C09150=1155.130,217.101,-63.506,-177.845,7.375,148.764
C09151=1155.134,216.851,-63.482,-177.849,7.372,148.764
C09152=1155.139,216.603,-63.456,-177.851,7.369,148.764
C09153=1155.143,216.355,-63.430,-177.854,7.367,148.765
C09154=1155.148,216.106,-63.406,-177.857,7.365,148.765
C09155=1155.152,215.857,-63.380,-177.860,7.362,148.765
C09156=1155.157,215.609,-63.356,-177.862,7.360,148.765
C09157=1155.161,215.360,-63.330,-177.865,7.357,148.765
C09158=1155.166,215.111,-63.306,-177.867,7.355,148.766
C09159=1155.170,214.862,-63.280,-177.871,7.352,148.766
C09160=1155.175,214.614,-63.256,-177.873,7.349,148.766
C09161=1155.179,214.364,-63.231,-177.876,7.347,148.766
C09162=1155.184,214.116,-63.205,-177.879,7.345,148.766
C09163=1155.188,213.867,-63.181,-177.881,7.343,148.767
C09164=1155.193,213.619,-63.156,-177.884,7.340,148.767
C09165=1155.197,213.370,-63.130,-177.887,7.337,148.767
C09166=1155.202,213.121,-63.106,-177.889,7.335,148.767
C09167=1155.206,212.873,-63.081,-177.893,7.332,148.767
C09168=1155.211,212.624,-63.056,-177.895,7.330,148.768
C09169=1155.216,212.375,-63.031,-177.898,7.328,148.768
C09170=1155.219,212.126,-63.006,-177.901,7.325,148.768
C09171=1155.225,211.878,-62.981,-177.903,7.323,148.768
C09172=1155.229,211.628,-62.956,-177.906,7.320,148.768
C09173=1155.233,211.381,-62.932,-177.908,7.318,148.768
C09174=1155.238,211.132,-62.907,-177.912,7.315,148.769
C09175=1155.242,210.883,-62.883,-177.914,7.312,148.769
C09176=1155.247,210.634,-62.858,-177.917,7.311,148.769
C09177=1155.251,210.385,-62.832,-177.920,7.308,148.769
C09178=1155.257,210.115,-62.805,-177.923,7.305,148.770
C09179=1155.261,209.844,-62.778,-177.925,7.303,148.770
C09180=1155.266,209.574,-62.752,-177.929,7.300,148.770
C09181=1155.272,209.303,-62.726,-177.931,7.298,148.770
C09182=1155.275,209.055,-62.700,-177.935,7.295,148.771
C09183=1155.280,208.806,-62.676,-177.937,7.293,148.771
C09184=1155.284,208.557,-62.651,-177.940,7.290,148.771
C09185=1155.289,208.308,-62.627,-177.942,7.288,148.771
C09186=1155.294,208.059,-62.602,-177.946,7.286,148.771
C09187=1155.298,207.810,-62.578,-177.948,7.283,148.771
C09188=1155.303,207.562,-62.553,-177.951,7.281,148.772
C09189=1155.308,207.313,-62.529,-177.954,7.278,148.772
C09190=1155.312,207.064,-62.503,-177.957,7.276,148.772
C09191=1155.316,206.816,-62.479,-177.959,7.273,148.772
C09192=1155.322,206.567,-62.454,-177.962,7.272,148.773
C09193=1155.325,206.318,-62.430,-177.965,7.269,148.773
C09194=1155.330,206.070,-62.406,-177.967,7.266,148.773
C09195=1155.335,205.821,-62.381,-177.970,7.264,148.773
C09196=1155.339,205.573,-62.357,-177.973,7.261,148.773
C09197=1155.344,205.323,-62.332,-177.976,7.259,148.774
C09198=1155.348,205.075,-62.308,-177.979,7.256,148.774
C09199=1155.353,204.826,-62.283,-177.981,7.255,148.774
C09200=1155.357,204.577,-62.259,-177.984,7.252,148.774
C09201=1155.363,204.328,-62.235,-177.987,7.250,148.775
C09202=1155.367,204.079,-62.211,-177.990,7.247,148.775
C09203=1155.371,203.831,-62.187,-177.992,7.245,148.775
C09204=1155.376,203.581,-62.162,-177.995,7.242,148.775
C09205=1155.380,203.333,-62.138,-177.998,7.240,148.776
C09206=1155.385,203.084,-62.114,-178.000,7.238,148.776
C09207=1155.390,202.836,-62.089,-178.003,7.236,148.776
C09208=1155.394,202.587,-62.064,-178.006,7.233,148.776
C09209=1155.398,202.338,-62.041,-178.009,7.231,148.776
C09210=1155.403,202.089,-62.016,-178.011,7.228,148.777
C09211=1155.408,201.840,-61.992,-178.014,7.226,148.777
C09212=1155.412,201.591,-61.968,-178.017,7.224,148.777
C09213=1155.417,201.343,-61.943,-178.020,7.222,148.777
C09214=1155.421,201.094,-61.920,-178.023,7.219,148.778
C09215=1155.426,200.845,-61.896,-178.025,7.217,148.778
C09216=1155.430,200.597,-61.872,-178.028,7.215,148.778
C09217=1155.435,200.347,-61.847,-178.030,7.212,148.778
C09218=1155.439,200.098,-61.823,-178.034,7.210,148.779
C09219=1155.444,199.850,-61.799,-178.036,7.208,148.779
C09220=1155.448,199.601,-61.775,-178.039,7.205,148.779
C09221=1155.453,199.353,-61.751,-178.041,7.203,148.779
C09222=1155.458,199.104,-61.727,-178.045,7.200,148.779
C09223=1155.462,198.855,-61.703,-178.047,7.198,148.780
C09224=1155.467,198.606,-61.679,-178.050,7.196,148.780
C09225=1155.471,198.357,-61.655,-178.052,7.194,148.780
C09226=1155.476,198.108,-61.631,-178.056,7.191,148.780
C09227=1155.481,197.859,-61.607,-178.058,7.189,148.781
C09228=1155.485,197.611,-61.583,-178.061,7.186,148.781
C09229=1155.490,197.363,-61.559,-178.064,7.185,148.781
C09230=1155.494,197.113,-61.535,-178.067,7.182,148.781
C09231=1155.499,196.864,-61.511,-178.069,7.180,148.782
C09232=1155.503,196.615,-61.487,-178.072,7.177,148.782
C09233=1155.508,196.367,-61.463,-178.075,7.175,148.782
C09234=1155.513,196.118,-61.440,-178.078,7.172,148.782
C09235=1155.517,195.869,-61.416,-178.080,7.171,148.783
C09236=1155.522,195.620,-61.393,-178.083,7.168,148.783
C09237=1155.526,195.372,-61.368,-178.086,7.166,148.783
C09238=1155.531,195.123,-61.345,-178.088,7.164,148.783
C09239=1155.535,194.874,-61.321,-178.091,7.161,148.784
C09240=1155.541,194.625,-61.297,-178.094,7.160,148.784
C09241=1155.544,194.376,-61.273,-178.097,7.157,148.784
C09242=1155.549,194.127,-61.249,-178.099,7.155,148.784
C09243=1155.554,193.878,-61.226,-178.103,7.152,148.785
C09244=1155.558,193.629,-61.202,-178.105,7.150,148.785
C09245=1155.563,193.380,-61.178,-178.108,7.148,148.785
C09246=1155.567,193.132,-61.154,-178.110,7.146,148.785
C09247=1155.572,192.883,-61.131,-178.114,7.143,148.786
C09248=1155.577,192.634,-61.108,-178.116,7.141,148.786
C09249=1155.581,192.385,-61.084,-178.118,7.139,148.786
C09250=1155.586,192.136,-61.060,-178.122,7.137,148.786
C09251=1155.590,191.887,-61.037,-178.124,7.135,148.787
C09252=1155.595,191.639,-61.013,-178.127,7.132,148.787
C09253=1155.600,191.390,-60.989,-178.130,7.130,148.787
C09254=1155.604,191.141,-60.966,-178.133,7.127,148.787
C09255=1155.609,190.892,-60.943,-178.135,7.125,148.788
C09256=1155.613,190.643,-60.919,-178.138,7.124,148.788
C09257=1155.618,190.394,-60.895,-178.141,7.121,148.788
C09258=1155.623,190.145,-60.872,-178.144,7.119,148.789
C09259=1155.627,189.896,-60.849,-178.146,7.116,148.789
C09260=1155.632,189.648,-60.824,-178.149,7.114,148.789
C09261=1155.636,189.399,-60.802,-178.152,7.112,148.789
C09262=1155.641,189.150,-60.778,-178.154,7.110,148.789
C09263=1155.645,188.901,-60.755,-178.157,7.108,148.790
C09264=1155.650,188.652,-60.732,-178.160,7.105,148.790
C09265=1155.655,188.403,-60.708,-178.163,7.103,148.790
C09266=1155.660,188.155,-60.685,-178.166,7.101,148.791
C09267=1155.664,187.906,-60.661,-178.169,7.099,148.791
C09268=1155.669,187.657,-60.638,-178.171,7.097,148.791
C09269=1155.673,187.409,-60.615,-178.174,7.094,148.791
C09270=1155.678,187.160,-60.592,-178.176,7.092,148.792
C09271=1155.682,186.911,-60.568,-178.180,7.090,148.792
C09272=1155.687,186.662,-60.545,-178.182,7.088,148.792
C09273=1155.692,186.413,-60.522,-178.184,7.086,148.792
C09274=1155.696,186.163,-60.498,-178.188,7.083,148.793
C09275=1155.700,185.915,-60.476,-178.190,7.081,148.793
C09276=1155.705,185.666,-60.452,-178.193,7.079,148.793
C09277=1155.710,185.417,-60.429,-178.196,7.077,148.794
C09278=1155.715,185.168,-60.406,-178.199,7.075,148.794
C09279=1155.719,184.920,-60.383,-178.201,7.072,148.794
C09280=1155.724,184.671,-60.360,-178.204,7.070,148.794
C09281=1155.728,184.422,-60.336,-178.207,7.068,148.795
C09282=1155.734,184.152,-60.311,-178.210,7.066,148.795
C09283=1155.738,183.883,-60.286,-178.213,7.063,148.795
C09284=1155.743,183.613,-60.261,-178.215,7.061,148.796
C09285=1155.749,183.343,-60.236,-178.219,7.059,148.796
C09286=1155.753,183.095,-60.213,-178.222,7.056,148.796
C09287=1155.757,182.846,-60.190,-178.224,7.054,148.796
C09288=1155.762,182.596,-60.167,-178.227,7.052,148.797
C09289=1155.767,182.347,-60.144,-178.230,7.050,148.797
C09290=1155.772,182.099,-60.122,-178.232,7.048,148.797
C09291=1155.776,181.850,-60.098,-178.235,7.046,148.798
C09292=1155.780,181.601,-60.075,-178.238,7.043,148.798
C09293=1155.785,181.352,-60.052,-178.241,7.042,148.798
C09294=1155.790,181.103,-60.029,-178.243,7.040,148.798
C09295=1155.795,180.855,-60.007,-178.247,7.037,148.799
C09296=1155.799,180.605,-59.984,-178.249,7.035,148.799
C09297=1155.804,180.356,-59.960,-178.251,7.033,148.799
C09298=1155.808,180.107,-59.938,-178.255,7.031,148.800
C09299=1155.813,179.858,-59.915,-178.257,7.029,148.800
C09300=1155.818,179.610,-59.893,-178.260,7.027,148.800
C09301=1155.822,179.361,-59.869,-178.263,7.024,148.800
C09302=1155.827,179.111,-59.847,-178.266,7.022,148.801
C09303=1155.831,178.863,-59.824,-178.269,7.020,148.801
C09304=1155.836,178.614,-59.801,-178.271,7.018,148.801
C09305=1155.841,178.365,-59.779,-178.274,7.016,148.802
C09306=1155.845,178.116,-59.755,-178.277,7.013,148.802
C09307=1155.849,177.867,-59.733,-178.279,7.011,148.802
C09308=1155.855,177.618,-59.710,-178.282,7.010,148.803
C09309=1155.859,177.370,-59.688,-178.285,7.007,148.803
C09310=1155.864,177.121,-59.664,-178.288,7.005,148.803
C09311=1155.869,176.872,-59.643,-178.290,7.003,148.803
C09312=1155.873,176.623,-59.619,-178.293,7.001,148.804
C09313=1155.878,176.374,-59.597,-178.296,6.999,148.804
C09314=1155.883,176.125,-59.574,-178.299,6.997,148.804
C09315=1155.887,175.876,-59.552,-178.301,6.995,148.805
C09316=1155.892,175.627,-59.529,-178.304,6.993,148.805
C09317=1155.896,175.377,-59.507,-178.307,6.991,148.805
C09318=1155.901,175.129,-59.484,-178.310,6.989,148.806
C09319=1155.906,174.880,-59.462,-178.312,6.986,148.806
C09320=1155.910,174.631,-59.438,-178.315,6.984,148.806
C09321=1155.915,174.382,-59.417,-178.318,6.983,148.807
C09322=1155.919,174.133,-59.394,-178.321,6.980,148.807
C09323=1155.924,173.884,-59.371,-178.323,6.978,148.807
C09324=1155.929,173.636,-59.349,-178.326,6.976,148.807
C09325=1155.934,173.386,-59.326,-178.329,6.974,148.808
C09326=1155.938,173.138,-59.304,-178.332,6.972,148.808
C09327=1155.943,172.889,-59.282,-178.334,6.970,148.808
C09328=1155.948,172.639,-59.259,-178.337,6.968,148.809
C09329=1155.952,172.391,-59.237,-178.340,6.966,148.809
C09330=1155.956,172.142,-59.215,-178.343,6.964,148.809
C09331=1155.962,171.893,-59.192,-178.346,6.962,148.810
C09332=1155.966,171.644,-59.170,-178.348,6.959,148.810
C09333=1155.970,171.395,-59.147,-178.351,6.957,148.810
C09334=1155.976,171.146,-59.125,-178.354,6.956,148.811
C09335=1155.980,170.897,-59.102,-178.356,6.954,148.811
C09336=1155.985,170.648,-59.081,-178.359,6.951,148.811
C09337=1155.990,170.399,-59.058,-178.362,6.949,148.811
C09338=1155.994,170.150,-59.035,-178.365,6.948,148.812
C09339=1155.999,169.901,-59.014,-178.367,6.946,148.812
C09340=1156.004,169.652,-58.991,-178.371,6.943,148.813
C09341=1156.008,169.403,-58.969,-178.373,6.941,148.813
C09342=1156.012,169.154,-58.947,-178.376,6.939,148.813
C09343=1156.017,168.906,-58.925,-178.378,6.938,148.813
C09344=1156.022,168.656,-58.902,-178.382,6.935,148.814
C09345=1156.027,168.407,-58.881,-178.384,6.933,148.814
C09346=1156.031,168.158,-58.859,-178.386,6.931,148.814
C09347=1156.036,167.909,-58.837,-178.390,6.929,148.815
C09348=1156.041,167.660,-58.813,-178.392,6.927,148.815
C09349=1156.045,167.411,-58.791,-178.395,6.925,148.815
C09350=1156.050,167.162,-58.770,-178.398,6.923,148.816
C09351=1156.054,166.913,-58.748,-178.401,6.921,148.816
C09352=1156.059,166.664,-58.726,-178.403,6.919,148.816
C09353=1156.064,166.415,-58.703,-178.406,6.917,148.817
C09354=1156.069,166.166,-58.682,-178.409,6.915,148.817
C09355=1156.074,165.918,-58.660,-178.412,6.913,148.817
C09356=1156.078,165.668,-58.638,-178.415,6.911,148.818
C09357=1156.083,165.420,-58.616,-178.417,6.909,148.818
C09358=1156.087,165.170,-58.594,-178.420,6.907,148.818
C09359=1156.092,164.922,-58.572,-178.422,6.905,148.819
C09360=1156.096,164.673,-58.550,-178.426,6.903,148.819
C09361=1156.102,164.424,-58.528,-178.428,6.901,148.819
C09362=1156.106,164.175,-58.505,-178.431,6.899,148.820
C09363=1156.111,163.925,-58.485,-178.433,6.897,148.820
C09364=1156.116,163.676,-58.462,-178.436,6.895,148.820
C09365=1156.120,163.427,-58.441,-178.439,6.893,148.821
C09366=1156.125,163.178,-58.419,-178.442,6.891,148.821
C09367=1156.130,162.929,-58.397,-178.445,6.890,148.821
C09368=1156.134,162.681,-58.375,-178.447,6.888,148.822
C09369=1156.139,162.431,-58.353,-178.451,6.885,148.822
C09370=1156.144,162.183,-58.332,-178.453,6.883,148.822
C09371=1156.148,161.933,-58.310,-178.455,6.881,148.823
C09372=1156.153,161.685,-58.288,-178.458,6.880,148.823
C09373=1156.158,161.436,-58.266,-178.461,6.877,148.823
C09374=1156.162,161.187,-58.244,-178.464,6.875,148.824
C09375=1156.167,160.937,-58.223,-178.467,6.874,148.824
C09376=1156.171,160.688,-58.201,-178.470,6.872,148.824
C09377=1156.176,160.439,-58.179,-178.472,6.870,148.825
C09378=1156.181,160.191,-58.158,-178.475,6.867,148.825
C09379=1156.185,159.942,-58.136,-178.478,6.866,148.825
C09380=1156.190,159.692,-58.115,-178.480,6.864,148.826
C09381=1156.195,159.443,-58.093,-178.483,6.862,148.826
C09382=1156.200,159.194,-58.071,-178.486,6.860,148.826
C09383=1156.204,158.946,-58.049,-178.489,6.859,148.827
C09384=1156.209,158.696,-58.028,-178.492,6.856,148.827
C09385=1156.214,158.447,-58.006,-178.494,6.854,148.827
C09386=1156.219,158.178,-57.984,-178.497,6.852,148.828
C09387=1156.224,157.909,-57.960,-178.500,6.850,148.828
C09388=1156.229,157.640,-57.937,-178.503,6.848,148.828
C09389=1156.234,157.371,-57.913,-178.506,6.846,148.829
C09390=1156.239,157.122,-57.892,-178.509,6.844,148.829
C09391=1156.244,156.874,-57.870,-178.511,6.842,148.830
C09392=1156.248,156.624,-57.849,-178.514,6.840,148.830
C09393=1156.252,156.375,-57.828,-178.517,6.839,148.830
C09394=1156.258,156.126,-57.807,-178.519,6.837,148.831
C09395=1156.263,155.877,-57.785,-178.523,6.834,148.831
C09396=1156.267,155.628,-57.763,-178.525,6.833,148.831
C09397=1156.272,155.379,-57.742,-178.528,6.831,148.832
C09398=1156.276,155.130,-57.721,-178.531,6.829,148.832
C09399=1156.281,154.881,-57.700,-178.534,6.827,148.833
C09400=1156.286,154.632,-57.678,-178.536,6.825,148.833
C09401=1156.291,154.383,-57.657,-178.539,6.823,148.833
C09402=1156.296,154.134,-57.635,-178.542,6.821,148.834
C09403=1156.300,153.885,-57.615,-178.544,6.819,148.834
C09404=1156.304,153.636,-57.593,-178.547,6.817,148.834
C09405=1156.309,153.386,-57.572,-178.550,6.816,148.835
C09406=1156.314,153.138,-57.550,-178.553,6.814,148.835
C09407=1156.319,152.888,-57.529,-178.555,6.812,148.835
C09408=1156.323,152.639,-57.508,-178.559,6.810,148.836
C09409=1156.328,152.390,-57.487,-178.561,6.808,148.836
C09410=1156.333,152.142,-57.465,-178.564,6.806,148.837
C09411=1156.337,151.893,-57.445,-178.567,6.805,148.837
C09412=1156.342,151.644,-57.423,-178.569,6.802,148.837
C09413=1156.347,151.394,-57.402,-178.572,6.801,148.837
C09414=1156.352,151.145,-57.381,-178.574,6.799,148.838
C09415=1156.356,150.896,-57.360,-178.578,6.796,148.838
C09416=1156.361,150.647,-57.339,-178.580,6.795,148.839
C09417=1156.367,150.398,-57.318,-178.583,6.793,148.839
C09418=1156.370,150.149,-57.296,-178.586,6.791,148.839
C09419=1156.375,149.900,-57.275,-178.588,6.790,148.840
C09420=1156.380,149.650,-57.254,-178.591,6.788,148.840
C09421=1156.385,149.402,-57.233,-178.594,6.786,148.840
C09422=1156.390,149.153,-57.212,-178.597,6.784,148.841
C09423=1156.395,148.903,-57.191,-178.599,6.783,148.841
C09424=1156.399,148.655,-57.170,-178.603,6.780,148.842
C09425=1156.404,148.405,-57.149,-178.605,6.778,148.842
C09426=1156.408,148.156,-57.128,-178.608,6.777,148.842
C09427=1156.413,147.907,-57.108,-178.611,6.775,148.843
C09428=1156.418,147.658,-57.086,-178.613,6.773,148.843
C09429=1156.423,147.409,-57.065,-178.616,6.771,148.844
C09430=1156.428,147.160,-57.044,-178.619,6.770,148.844
C09431=1156.432,146.911,-57.024,-178.621,6.768,148.844
C09432=1156.437,146.662,-57.003,-178.624,6.766,148.844
C09433=1156.441,146.413,-56.982,-178.626,6.764,148.845
C09434=1156.446,146.164,-56.961,-178.630,6.762,148.845
C09435=1156.451,145.915,-56.940,-178.632,6.760,148.846
C09436=1156.456,145.665,-56.919,-178.635,6.758,148.846
C09437=1156.461,145.416,-56.898,-178.638,6.756,148.846
C09438=1156.465,145.167,-56.878,-178.640,6.755,148.847
C09439=1156.470,144.918,-56.857,-178.643,6.753,148.847
C09440=1156.475,144.669,-56.837,-178.646,6.751,148.848
C09441=1156.480,144.420,-56.816,-178.649,6.750,148.848
C09442=1156.484,144.171,-56.795,-178.651,6.748,148.848
C09443=1156.489,143.922,-56.774,-178.654,6.746,148.849
C09444=1156.494,143.673,-56.753,-178.657,6.744,148.849
C09445=1156.498,143.424,-56.733,-178.659,6.743,148.849
C09446=1156.503,143.175,-56.712,-178.663,6.740,148.850
C09447=1156.508,142.926,-56.692,-178.665,6.738,148.850
C09448=1156.513,142.677,-56.671,-178.668,6.737,148.851
C09449=1156.517,142.427,-56.650,-178.671,6.735,148.851
C09450=1156.521,142.178,-56.630,-178.674,6.733,148.851
C09451=1156.527,141.929,-56.609,-178.676,6.731,148.852
C09452=1156.531,141.680,-56.588,-178.679,6.730,148.852
C09453=1156.536,141.431,-56.567,-178.682,6.728,148.853
C09454=1156.541,141.182,-56.547,-178.684,6.726,148.853
C09455=1156.545,140.932,-56.527,-178.687,6.725,148.853
C09456=1156.550,140.683,-56.506,-178.690,6.723,148.854
C09457=1156.555,140.434,-56.486,-178.693,6.721,148.854
C09458=1156.560,140.185,-56.465,-178.695,6.719,148.854
C09459=1156.565,139.936,-56.445,-178.698,6.718,148.855
C09460=1156.570,139.688,-56.425,-178.701,6.716,148.855
C09461=1156.575,139.438,-56.404,-178.703,6.714,148.856
C09462=1156.579,139.189,-56.383,-178.706,6.713,148.856
C09463=1156.584,138.940,-56.364,-178.709,6.711,148.856
C09464=1156.589,138.691,-56.343,-178.712,6.708,148.857
C09465=1156.594,138.442,-56.322,-178.715,6.707,148.857
C09466=1156.598,138.193,-56.302,-178.717,6.705,148.858
C09467=1156.602,137.944,-56.281,-178.720,6.703,148.858
C09468=1156.608,137.694,-56.261,-178.723,6.701,148.858
C09469=1156.612,137.445,-56.241,-178.726,6.700,148.859
C09470=1156.617,137.196,-56.220,-178.729,6.698,148.859
C09471=1156.621,136.947,-56.200,-178.731,6.697,148.860
C09472=1156.627,136.697,-56.180,-178.734,6.695,148.860
C09473=1156.631,136.448,-56.159,-178.737,6.693,148.861
C09474=1156.636,136.199,-56.139,-178.740,6.691,148.861
C09475=1156.641,135.951,-56.119,-178.742,6.690,148.861
C09476=1156.646,135.701,-56.099,-178.745,6.688,148.862
C09477=1156.650,135.452,-56.078,-178.748,6.686,148.862
C09478=1156.655,135.203,-56.058,-178.750,6.685,148.862
C09479=1156.660,134.954,-56.038,-178.753,6.683,148.863
C09480=1156.664,134.705,-56.018,-178.756,6.681,148.863
C09481=1156.669,134.455,-55.997,-178.759,6.679,148.864
C09482=1156.674,134.206,-55.977,-178.761,6.678,148.864
C09483=1156.679,133.958,-55.957,-178.764,6.676,148.864
C09484=1156.684,133.708,-55.938,-178.767,6.674,148.865
C09485=1156.688,133.459,-55.917,-178.769,6.672,148.865
C09486=1156.693,133.210,-55.896,-178.772,6.671,148.866
C09487=1156.698,132.960,-55.877,-178.775,6.669,148.866
C09488=1156.703,132.711,-55.856,-178.778,6.667,148.866
C09489=1156.708,132.462,-55.837,-178.780,6.666,148.867
C09490=1156.713,132.194,-55.815,-178.783,6.664,148.867
C09491=1156.718,131.925,-55.794,-178.786,6.663,148.868
C09492=1156.723,131.657,-55.773,-178.789,6.661,148.868
C09493=1156.728,131.388,-55.750,-178.792,6.658,148.869
C09494=1156.733,131.139,-55.730,-178.795,6.657,148.869
C09495=1156.738,130.889,-55.711,-178.798,6.655,148.870
C09496=1156.742,130.640,-55.690,-178.801,6.653,148.870
C09497=1156.747,130.391,-55.671,-178.804,6.652,148.870
C09498=1156.752,130.143,-55.651,-178.806,6.650,148.871
C09499=1156.757,129.893,-55.631,-178.809,6.648,148.871
C09500=1156.761,129.644,-55.611,-178.812,6.647,148.872
C09501=1156.766,129.394,-55.591,-178.814,6.645,148.872
C09502=1156.771,129.146,-55.572,-178.816,6.644,148.872
C09503=1156.776,128.897,-55.551,-178.819,6.642,148.873
C09504=1156.781,128.647,-55.532,-178.822,6.641,148.873
C09505=1156.785,128.398,-55.511,-178.825,6.639,148.874
C09506=1156.790,128.149,-55.492,-178.827,6.637,148.874
C09507=1156.795,127.900,-55.472,-178.831,6.636,148.875
C09508=1156.800,127.651,-55.452,-178.833,6.634,148.875
C09509=1156.804,127.401,-55.432,-178.836,6.632,148.875
C09510=1156.810,127.152,-55.413,-178.839,6.631,148.876
C09511=1156.814,126.903,-55.393,-178.841,6.629,148.876
C09512=1156.819,126.654,-55.373,-178.844,6.627,148.877
C09513=1156.824,126.405,-55.354,-178.847,6.625,148.877
C09514=1156.829,126.155,-55.334,-178.850,6.624,148.877
C09515=1156.833,125.906,-55.314,-178.852,6.622,148.878
C09516=1156.838,125.657,-55.294,-178.855,6.620,148.878
C09517=1156.843,125.408,-55.275,-178.858,6.619,148.879
C09518=1156.848,125.158,-55.255,-178.861,6.617,148.879
C09519=1156.852,124.910,-55.235,-178.864,6.616,148.880
C09520=1156.857,124.661,-55.216,-178.866,6.614,148.880
C09521=1156.862,124.411,-55.196,-178.868,6.613,148.880
C09522=1156.867,124.162,-55.177,-178.871,6.611,148.881
C09523=1156.872,123.913,-55.158,-178.874,6.609,148.881
C09524=1156.877,123.664,-55.137,-178.877,6.608,148.882
C09525=1156.881,123.414,-55.118,-178.879,6.606,148.882
C09526=1156.887,123.165,-55.098,-178.882,6.605,148.883
C09527=1156.891,122.916,-55.079,-178.885,6.603,148.883
C09528=1156.895,122.667,-55.059,-178.888,6.601,148.883
C09529=1156.901,122.418,-55.040,-178.891,6.600,148.884
C09530=1156.905,122.168,-55.021,-178.893,6.598,148.884
C09531=1156.910,121.919,-55.001,-178.896,6.596,148.885
C09532=1156.915,121.670,-54.982,-178.899,6.594,148.885
C09533=1156.920,121.421,-54.963,-178.901,6.593,148.885
C09534=1156.925,121.172,-54.943,-178.904,6.592,148.886
C09535=1156.929,120.923,-54.923,-178.907,6.590,148.886
C09536=1156.934,120.673,-54.903,-178.910,6.589,148.887
C09537=1156.939,120.425,-54.885,-178.912,6.587,148.887
C09538=1156.943,120.175,-54.865,-178.915,6.585,148.888
C09539=1156.949,119.926,-54.846,-178.918,6.584,148.888
C09540=1156.953,119.677,-54.826,-178.920,6.582,148.888
C09541=1156.957,119.427,-54.807,-178.924,6.581,148.889
C09542=1156.963,119.178,-54.788,-178.926,6.579,148.889
C09543=1156.968,118.928,-54.769,-178.929,6.577,148.890
C09544=1156.972,118.680,-54.750,-178.931,6.576,148.890
C09545=1156.977,118.430,-54.730,-178.934,6.575,148.891
C09546=1156.983,118.181,-54.711,-178.937,6.573,148.891
C09547=1156.987,117.932,-54.691,-178.940,6.571,148.892
C09548=1156.992,117.683,-54.673,-178.943,6.570,148.892
C09549=1156.997,117.434,-54.653,-178.945,6.568,148.892
C09550=1157.002,117.185,-54.634,-178.948,6.566,148.893
C09551=1157.006,116.935,-54.615,-178.951,6.565,148.893
C09552=1157.011,116.686,-54.595,-178.953,6.564,148.894
C09553=1157.016,116.436,-54.576,-178.956,6.562,148.894
C09554=1157.020,116.187,-54.557,-178.959,6.561,148.895
C09555=1157.026,115.938,-54.538,-178.961,6.559,148.895
C09556=1157.031,115.689,-54.518,-178.964,6.557,148.896
C09557=1157.035,115.440,-54.500,-178.967,6.556,148.896
C09558=1157.040,115.190,-54.481,-178.970,6.554,148.896
C09559=1157.045,114.941,-54.462,-178.972,6.552,148.897
C09560=1157.050,114.692,-54.442,-178.975,6.552,148.897
C09561=1157.055,114.443,-54.423,-178.978,6.550,148.898
C09562=1157.059,114.194,-54.404,-178.980,6.548,148.898
C09563=1157.065,113.944,-54.385,-178.983,6.547,148.899
C09564=1157.069,113.696,-54.367,-178.986,6.545,148.899
C09565=1157.074,113.446,-54.347,-178.989,6.543,148.900
C09566=1157.079,113.197,-54.329,-178.992,6.542,148.900
C09567=1157.084,112.947,-54.309,-178.994,6.541,148.900
C09568=1157.089,112.698,-54.290,-178.997,6.539,148.901
C09569=1157.093,112.449,-54.272,-178.999,6.537,148.901
C09570=1157.099,112.200,-54.253,-179.002,6.536,148.902
C09571=1157.103,111.950,-54.234,-179.005,6.534,148.902
C09572=1157.108,111.701,-54.215,-179.008,6.533,148.903
C09573=1157.113,111.452,-54.196,-179.010,6.532,148.903
C09574=1157.118,111.203,-54.177,-179.013,6.530,148.904
C09575=1157.122,110.954,-54.159,-179.016,6.528,148.904
C09576=1157.127,110.704,-54.139,-179.019,6.527,148.905
C09577=1157.132,110.455,-54.121,-179.021,6.525,148.905
C09578=1157.137,110.206,-54.102,-179.024,6.524,148.905
C09579=1157.141,109.957,-54.083,-179.026,6.523,148.906
C09580=1157.146,109.708,-54.065,-179.029,6.521,148.906
C09581=1157.151,109.458,-54.045,-179.032,6.520,148.907
C09582=1157.156,109.209,-54.027,-179.035,6.518,148.907
C09583=1157.161,108.960,-54.008,-179.038,6.516,148.908
C09584=1157.166,108.710,-53.989,-179.040,6.515,148.908
C09585=1157.171,108.461,-53.970,-179.043,6.514,148.908
C09586=1157.176,108.212,-53.952,-179.046,6.512,148.909
C09587=1157.180,107.963,-53.933,-179.048,6.511,148.910
C09588=1157.186,107.713,-53.914,-179.051,6.509,148.910
C09589=1157.190,107.464,-53.895,-179.054,6.507,148.910
C09590=1157.195,107.215,-53.877,-179.056,6.506,148.911
C09591=1157.200,106.966,-53.858,-179.059,6.505,148.911
C09592=1157.204,106.716,-53.840,-179.062,6.503,148.912
C09593=1157.210,106.467,-53.821,-179.065,6.502,148.912
C09594=1157.215,106.199,-53.801,-179.068,6.500,148.913
C09595=1157.220,105.931,-53.781,-179.071,6.499,148.913
C09596=1157.225,105.662,-53.761,-179.073,6.497,148.914
C09597=1157.230,105.394,-53.741,-179.077,6.496,148.914
C09598=1157.235,105.144,-53.723,-179.079,6.494,148.915
C09599=1157.240,104.895,-53.705,-179.081,6.493,148.915
C09600=1157.245,104.646,-53.685,-179.084,6.491,148.916
C09601=1157.250,104.397,-53.667,-179.087,6.490,148.916
C09602=1157.255,104.147,-53.649,-179.090,6.488,148.917
C09603=1157.259,103.898,-53.630,-179.093,6.487,148.917
C09604=1157.264,103.649,-53.611,-179.095,6.486,148.917
C09605=1157.269,103.399,-53.593,-179.098,6.484,148.918
C09606=1157.274,103.151,-53.575,-179.101,6.483,148.918
C09607=1157.279,102.901,-53.556,-179.104,6.481,148.919
C09608=1157.284,102.652,-53.538,-179.106,6.480,148.919
C09609=1157.289,102.402,-53.520,-179.108,6.478,148.920
C09610=1157.293,102.154,-53.501,-179.112,6.477,148.920
C09611=1157.298,101.904,-53.483,-179.114,6.475,148.921
C09612=1157.303,101.654,-53.464,-179.117,6.474,148.921
C09613=1157.308,101.405,-53.446,-179.119,6.473,148.922
C09614=1157.313,101.156,-53.428,-179.122,6.471,148.922
C09615=1157.317,100.907,-53.409,-179.125,6.470,148.923
C09616=1157.323,100.657,-53.391,-179.128,6.468,148.923
C09617=1157.328,100.408,-53.373,-179.130,6.467,148.923
C09618=1157.333,100.159,-53.355,-179.133,6.466,148.924
C09619=1157.337,99.909,-53.336,-179.136,6.464,148.924
C09620=1157.342,99.660,-53.318,-179.139,6.462,148.925
C09621=1157.347,99.411,-53.300,-179.141,6.461,148.925
C09622=1157.351,99.162,-53.282,-179.144,6.460,148.926
C09623=1157.357,98.913,-53.263,-179.147,6.458,148.926
C09624=1157.361,98.663,-53.245,-179.149,6.457,148.927
C09625=1157.366,98.414,-53.227,-179.152,6.456,148.927
C09626=1157.371,98.164,-53.209,-179.155,6.454,148.928
C09627=1157.376,97.915,-53.191,-179.158,6.453,148.928
C09628=1157.381,97.666,-53.173,-179.160,6.451,148.929
C09629=1157.386,97.417,-53.155,-179.163,6.451,148.929
C09630=1157.390,97.167,-53.136,-179.166,6.449,148.930
C09631=1157.395,96.918,-53.118,-179.168,6.447,148.930
C09632=1157.401,96.668,-53.100,-179.171,6.445,148.931
C09633=1157.406,96.419,-53.082,-179.174,6.445,148.931
C09634=1157.411,96.170,-53.064,-179.176,6.443,148.932
C09635=1157.416,95.921,-53.046,-179.179,6.442,148.932
C09636=1157.420,95.672,-53.028,-179.181,6.441,148.932
C09637=1157.425,95.422,-53.010,-179.184,6.439,148.933
C09638=1157.430,95.173,-52.992,-179.187,6.438,148.934
C09639=1157.435,94.923,-52.974,-179.190,6.436,148.934
C09640=1157.440,94.674,-52.956,-179.193,6.435,148.935
C09641=1157.444,94.425,-52.938,-179.195,6.434,148.935
C09642=1157.449,94.176,-52.920,-179.198,6.432,148.935
C09643=1157.454,93.927,-52.902,-179.200,6.431,148.936
C09644=1157.459,93.678,-52.884,-179.203,6.430,148.936
C09645=1157.464,93.428,-52.867,-179.206,6.428,148.937
C09646=1157.469,93.179,-52.849,-179.209,6.426,148.937
C09647=1157.474,92.929,-52.830,-179.211,6.426,148.938
C09648=1157.479,92.680,-52.812,-179.214,6.424,148.938
C09649=1157.483,92.430,-52.794,-179.217,6.423,148.939
C09650=1157.488,92.181,-52.776,-179.219,6.422,148.939
C09651=1157.494,91.931,-52.759,-179.222,6.420,148.940
C09652=1157.498,91.682,-52.741,-179.225,6.419,148.940
C09653=1157.503,91.433,-52.723,-179.227,6.418,148.941
C09654=1157.508,91.184,-52.706,-179.230,6.416,148.941
C09655=1157.512,90.935,-52.688,-179.233,6.415,148.942
C09656=1157.518,90.685,-52.670,-179.236,6.413,148.942
C09657=1157.523,90.436,-52.652,-179.238,6.412,148.943
C09658=1157.528,90.187,-52.634,-179.241,6.411,148.943
C09659=1157.532,89.938,-52.616,-179.244,6.409,148.944
C09660=1157.538,89.688,-52.599,-179.246,6.408,148.944
C09661=1157.543,89.439,-52.581,-179.249,6.407,148.945
C09662=1157.547,89.190,-52.563,-179.252,6.405,148.945
C09663=1157.552,88.940,-52.547,-179.254,6.404,148.946
C09664=1157.557,88.691,-52.529,-179.257,6.403,148.946
C09665=1157.562,88.442,-52.511,-179.260,6.401,148.947
C09666=1157.567,88.192,-52.493,-179.262,6.401,148.947
C09667=1157.572,87.943,-52.475,-179.265,6.399,148.948
C09668=1157.577,87.694,-52.457,-179.268,6.398,148.948
C09669=1157.581,87.444,-52.441,-179.270,6.397,148.949
C09670=1157.586,87.195,-52.423,-179.273,6.395,148.949
C09671=1157.591,86.946,-52.405,-179.276,6.394,148.950
C09672=1157.596,86.696,-52.387,-179.278,6.393,148.950
C09673=1157.601,86.447,-52.369,-179.281,6.391,148.951
C09674=1157.606,86.197,-52.353,-179.284,6.390,148.951
C09675=1157.611,85.948,-52.335,-179.286,6.389,148.952
C09676=1157.616,85.699,-52.317,-179.289,6.387,148.952
C09677=1157.621,85.449,-52.300,-179.292,6.386,148.953
C09678=1157.625,85.200,-52.282,-179.295,6.385,148.953
C09679=1157.630,84.950,-52.265,-179.297,6.383,148.953
C09680=1157.635,84.701,-52.247,-179.300,6.382,148.954
C09681=1157.640,84.452,-52.230,-179.303,6.381,148.955
C09682=1157.645,84.203,-52.213,-179.305,6.379,148.955
C09683=1157.650,83.954,-52.195,-179.309,6.378,148.956
C09684=1157.655,83.704,-52.177,-179.311,6.377,148.956
C09685=1157.660,83.455,-52.161,-179.313,6.376,148.956
C09686=1157.665,83.206,-52.143,-179.316,6.375,148.957
C09687=1157.670,82.956,-52.126,-179.319,6.373,148.958
C09688=1157.675,82.706,-52.108,-179.322,6.372,148.958
C09689=1157.679,82.457,-52.091,-179.324,6.371,148.959
C09690=1157.684,82.207,-52.074,-179.327,6.369,148.959
C09691=1157.689,81.958,-52.056,-179.330,6.368,148.959
C09692=1157.694,81.710,-52.039,-179.332,6.367,148.960
C09693=1157.699,81.460,-52.021,-179.335,6.366,148.961
C09694=1157.704,81.211,-52.005,-179.337,6.365,148.961
C09695=1157.709,80.961,-51.987,-179.340,6.363,148.962
C09696=1157.714,80.712,-51.969,-179.343,6.362,148.962
C09697=1157.718,80.462,-51.953,-179.345,6.361,148.963
C09698=1157.724,80.194,-51.934,-179.348,6.359,148.963
C09699=1157.730,79.925,-51.916,-179.351,6.358,148.964
C09700=1157.734,79.657,-51.897,-179.354,6.356,148.964
C09701=1157.740,79.389,-51.879,-179.357,6.355,148.965
C09702=1157.745,79.139,-51.861,-179.360,6.354,148.965
C09703=1157.750,78.890,-51.845,-179.363,6.353,148.966
C09704=1157.755,78.641,-51.827,-179.365,6.352,148.966
C09705=1157.759,78.391,-51.810,-179.368,6.350,148.967
C09706=1157.765,78.142,-51.793,-179.371,6.349,148.967
C09707=1157.770,77.893,-51.776,-179.373,6.348,148.968
C09708=1157.774,77.644,-51.758,-179.376,6.347,148.968
C09709=1157.780,77.394,-51.741,-179.378,6.346,148.969
C09710=1157.784,77.144,-51.725,-179.381,6.344,148.969
C09711=1157.790,76.895,-51.708,-179.384,6.343,148.970
C09712=1157.794,76.646,-51.691,-179.386,6.342,148.970
C09713=1157.799,76.397,-51.673,-179.389,6.340,148.971
C09714=1157.804,76.147,-51.656,-179.392,6.340,148.971
C09715=1157.810,75.898,-51.639,-179.394,6.338,148.972
C09716=1157.814,75.648,-51.623,-179.398,6.337,148.972
C09717=1157.819,75.399,-51.606,-179.400,6.336,148.973
C09718=1157.824,75.149,-51.589,-179.403,6.334,148.974
C09719=1157.829,74.900,-51.571,-179.405,6.334,148.974
C09720=1157.834,74.651,-51.555,-179.408,6.332,148.974
C09721=1157.838,74.402,-51.538,-179.410,6.331,148.975
C09722=1157.844,74.152,-51.521,-179.413,6.330,148.975
C09723=1157.849,73.903,-51.504,-179.416,6.328,148.976
C09724=1157.854,73.653,-51.487,-179.419,6.328,148.977
C09725=1157.858,73.404,-51.470,-179.421,6.326,148.977
C09726=1157.863,73.154,-51.453,-179.423,6.325,148.977
C09727=1157.869,72.905,-51.437,-179.427,6.324,148.978
C09728=1157.873,72.656,-51.420,-179.429,6.323,148.978
C09729=1157.878,72.406,-51.403,-179.432,6.321,148.979
C09730=1157.883,72.157,-51.386,-179.435,6.320,148.980
C09731=1157.889,71.907,-51.369,-179.437,6.319,148.980
C09732=1157.893,71.658,-51.353,-179.440,6.318,148.981
C09733=1157.898,71.408,-51.336,-179.442,6.317,148.981
C09734=1157.903,71.159,-51.319,-179.445,6.315,148.982
C09735=1157.908,70.910,-51.302,-179.448,6.315,148.982
C09736=1157.912,70.660,-51.286,-179.450,6.313,148.983
C09737=1157.918,70.411,-51.269,-179.453,6.312,148.983
C09738=1157.923,70.162,-51.252,-179.456,6.311,148.984
C09739=1157.927,69.912,-51.235,-179.458,6.310,148.984
C09740=1157.933,69.663,-51.219,-179.461,6.309,148.985
C09741=1157.937,69.414,-51.202,-179.464,6.307,148.985
C09742=1157.942,69.164,-51.185,-179.466,6.306,148.986
C09743=1157.948,68.915,-51.168,-179.469,6.305,148.986
C09744=1157.952,68.666,-51.152,-179.471,6.304,148.987
C09745=1157.957,68.416,-51.136,-179.475,6.303,148.987
C09746=1157.963,68.167,-51.119,-179.477,6.302,148.988
C09747=1157.967,67.917,-51.102,-179.480,6.300,148.989
C09748=1157.972,67.668,-51.086,-179.482,6.299,148.989
C09749=1157.977,67.419,-51.069,-179.485,6.298,148.989
C09750=1157.982,67.169,-51.052,-179.487,6.297,148.990
C09751=1157.987,66.920,-51.036,-179.490,6.296,148.990
C09752=1157.992,66.670,-51.020,-179.493,6.295,148.991
C09753=1157.997,66.421,-51.003,-179.496,6.293,148.992
C09754=1158.002,66.171,-50.986,-179.498,6.293,148.992
C09755=1158.007,65.922,-50.969,-179.501,6.291,148.993
C09756=1158.012,65.673,-50.954,-179.503,6.290,148.993
C09757=1158.017,65.423,-50.937,-179.506,6.289,148.994
C09758=1158.022,65.174,-50.921,-179.509,6.287,148.994
C09759=1158.027,64.925,-50.904,-179.511,6.287,148.995
C09760=1158.032,64.674,-50.888,-179.514,6.285,148.995
C09761=1158.037,64.426,-50.871,-179.517,6.284,148.996
C09762=1158.041,64.176,-50.855,-179.520,6.283,148.996
C09763=1158.047,63.927,-50.839,-179.522,6.282,148.997
C09764=1158.051,63.677,-50.822,-179.525,6.281,148.997
C09765=1158.057,63.428,-50.806,-179.527,6.280,148.998
C09766=1158.061,63.179,-50.789,-179.530,6.278,148.998
C09767=1158.067,62.929,-50.773,-179.533,6.278,148.999
C09768=1158.071,62.680,-50.757,-179.535,6.276,148.999
C09769=1158.076,62.430,-50.741,-179.538,6.275,149.000
C09770=1158.081,62.181,-50.724,-179.541,6.274,149.001
C09771=1158.086,61.931,-50.708,-179.543,6.273,149.001
C09772=1158.091,61.682,-50.692,-179.546,6.272,149.002
C09773=1158.096,61.432,-50.675,-179.548,6.271,149.002
C09774=1158.101,61.183,-50.659,-179.552,6.270,149.003
C09775=1158.106,60.933,-50.643,-179.554,6.269,149.003
C09776=1158.111,60.685,-50.626,-179.556,6.268,149.004
C09777=1158.116,60.434,-50.610,-179.559,6.267,149.004
C09778=1158.121,60.186,-50.594,-179.561,6.266,149.005
C09779=1158.126,59.936,-50.578,-179.565,6.265,149.005
C09780=1158.131,59.687,-50.562,-179.567,6.264,149.006
C09781=1158.136,59.437,-50.546,-179.569,6.262,149.006
C09782=1158.141,59.188,-50.529,-179.572,6.262,149.007
C09783=1158.146,58.939,-50.514,-179.575,6.260,149.007
C09784=1158.151,58.689,-50.497,-179.577,6.259,149.008
C09785=1158.156,58.440,-50.482,-179.580,6.258,149.008
C09786=1158.160,58.190,-50.465,-179.583,6.257,149.009
C09787=1158.166,57.941,-50.449,-179.586,6.256,149.010
C09788=1158.170,57.691,-50.433,-179.588,6.255,149.010
C09789=1158.176,57.442,-50.417,-179.591,6.253,149.011
C09790=1158.180,57.192,-50.400,-179.593,6.253,149.011
C09791=1158.186,56.943,-50.385,-179.596,6.251,149.012
C09792=1158.191,56.694,-50.369,-179.598,6.250,149.012
C09793=1158.195,56.444,-50.353,-179.601,6.250,149.013
C09794=1158.201,56.195,-50.337,-179.604,6.248,149.013
C09795=1158.205,55.945,-50.320,-179.606,6.247,149.014
C09796=1158.211,55.696,-50.305,-179.609,6.246,149.014
C09797=1158.215,55.446,-50.289,-179.611,6.245,149.015
C09798=1158.221,55.197,-50.273,-179.615,6.244,149.016
C09799=1158.226,54.948,-50.257,-179.617,6.243,149.016
C09800=1158.230,54.698,-50.240,-179.620,6.242,149.017
C09801=1158.236,54.449,-50.225,-179.622,6.241,149.017
C09802=1158.241,54.180,-50.208,-179.625,6.240,149.018
C09803=1158.246,53.911,-50.190,-179.628,6.239,149.018
C09804=1158.252,53.642,-50.173,-179.631,6.237,149.019
C09805=1158.257,53.374,-50.156,-179.633,6.237,149.020
C09806=1158.262,53.125,-50.141,-179.636,6.235,149.020
C09807=1158.267,52.875,-50.125,-179.638,6.234,149.020
C09808=1158.272,52.626,-50.109,-179.642,6.233,149.021
C09809=1158.277,52.377,-50.093,-179.644,6.232,149.021
C09810=1158.282,52.127,-50.077,-179.647,6.231,149.022
C09811=1158.287,51.878,-50.061,-179.649,6.230,149.023
C09812=1158.293,51.628,-50.046,-179.652,6.230,149.023
C09813=1158.297,51.379,-50.030,-179.654,6.228,149.024
C09814=1158.302,51.129,-50.015,-179.657,6.228,149.024
C09815=1158.307,50.880,-49.999,-179.660,6.226,149.025
C09816=1158.312,50.630,-49.982,-179.662,6.225,149.025
C09817=1158.317,50.381,-49.967,-179.665,6.224,149.026
C09818=1158.322,50.132,-49.952,-179.667,6.223,149.026
C09819=1158.327,49.882,-49.936,-179.670,6.222,149.027
C09820=1158.332,49.632,-49.920,-179.673,6.221,149.027
C09821=1158.338,49.383,-49.905,-179.675,6.220,149.028
C09822=1158.342,49.133,-49.888,-179.678,6.219,149.029
C09823=1158.347,48.884,-49.873,-179.681,6.218,149.029
C09824=1158.352,48.635,-49.857,-179.683,6.217,149.030
C09825=1158.357,48.385,-49.842,-179.686,6.216,149.030
C09826=1158.362,48.135,-49.826,-179.688,6.215,149.031
C09827=1158.367,47.886,-49.811,-179.692,6.214,149.031
C09828=1158.372,47.637,-49.795,-179.694,6.213,149.032
C09829=1158.377,47.387,-49.779,-179.696,6.212,149.032
C09830=1158.382,47.137,-49.764,-179.699,6.211,149.033
C09831=1158.387,46.888,-49.749,-179.701,6.210,149.033
C09832=1158.392,46.639,-49.733,-179.705,6.209,149.034
C09833=1158.397,46.389,-49.717,-179.707,6.208,149.035
C09834=1158.402,46.140,-49.702,-179.709,6.207,149.035
C09835=1158.407,45.890,-49.687,-179.712,6.206,149.036
C09836=1158.413,45.641,-49.671,-179.715,6.205,149.036
C09837=1158.417,45.391,-49.656,-179.717,6.204,149.037
C09838=1158.422,45.142,-49.640,-179.720,6.203,149.037
C09839=1158.427,44.892,-49.624,-179.722,6.202,149.038
C09840=1158.432,44.643,-49.610,-179.725,6.201,149.039
C09841=1158.438,44.394,-49.594,-179.728,6.200,149.039
C09842=1158.442,44.144,-49.578,-179.730,6.199,149.040
C09843=1158.447,43.895,-49.563,-179.733,6.198,149.040
C09844=1158.452,43.645,-49.547,-179.735,6.197,149.041
C09845=1158.458,43.396,-49.532,-179.738,6.197,149.041
C09846=1158.462,43.147,-49.517,-179.741,6.195,149.042
C09847=1158.467,42.897,-49.501,-179.743,6.194,149.042
C09848=1158.472,42.648,-49.486,-179.746,6.193,149.043
C09849=1158.477,42.398,-49.470,-179.749,6.192,149.044
C09850=1158.483,42.148,-49.455,-179.751,6.191,149.044
C09851=1158.488,41.899,-49.440,-179.754,6.190,149.045
C09852=1158.492,41.649,-49.424,-179.756,6.189,149.045
C09853=1158.497,41.400,-49.409,-179.759,6.189,149.046
C09854=1158.502,41.150,-49.394,-179.762,6.187,149.046
C09855=1158.507,40.901,-49.379,-179.764,6.187,149.047
C09856=1158.513,40.651,-49.364,-179.766,6.186,149.047
C09857=1158.518,40.402,-49.348,-179.770,6.185,149.048
C09858=1158.523,40.153,-49.333,-179.772,6.184,149.048
C09859=1158.528,39.903,-49.317,-179.774,6.183,149.049
C09860=1158.532,39.654,-49.302,-179.777,6.182,149.050
C09861=1158.538,39.404,-49.288,-179.779,6.181,149.050
C09862=1158.543,39.154,-49.273,-179.783,6.179,149.051
C09863=1158.548,38.905,-49.257,-179.785,6.179,149.051
C09864=1158.553,38.656,-49.242,-179.787,6.178,149.052
C09865=1158.558,38.406,-49.227,-179.790,6.176,149.052
C09866=1158.563,38.157,-49.212,-179.793,6.176,149.053
C09867=1158.568,37.907,-49.196,-179.795,6.175,149.053
C09868=1158.572,37.658,-49.181,-179.798,6.174,149.054
C09869=1158.578,37.408,-49.166,-179.800,6.173,149.055
C09870=1158.583,37.159,-49.151,-179.803,6.173,149.055
C09871=1158.588,36.909,-49.136,-179.805,6.172,149.056
C09872=1158.593,36.659,-49.121,-179.808,6.170,149.056
C09873=1158.598,36.410,-49.106,-179.811,6.170,149.057
C09874=1158.603,36.161,-49.091,-179.813,6.169,149.057
C09875=1158.608,35.911,-49.077,-179.816,6.167,149.058
C09876=1158.613,35.662,-49.061,-179.819,6.167,149.059
C09877=1158.618,35.412,-49.047,-179.821,6.166,149.059
C09878=1158.624,35.163,-49.031,-179.824,6.165,149.060
C09879=1158.628,34.914,-49.016,-179.826,6.164,149.060
C09880=1158.634,34.664,-49.001,-179.829,6.164,149.061
C09881=1158.639,34.415,-48.986,-179.832,6.162,149.061
C09882=1158.643,34.164,-48.972,-179.834,6.161,149.062
C09883=1158.648,33.915,-48.956,-179.836,6.161,149.062
C09884=1158.653,33.666,-48.941,-179.840,6.159,149.063
C09885=1158.658,33.416,-48.927,-179.842,6.158,149.063
C09886=1158.663,33.167,-48.911,-179.844,6.158,149.064
C09887=1158.668,32.917,-48.897,-179.847,6.157,149.065
C09888=1158.674,32.667,-48.881,-179.850,6.156,149.065
C09889=1158.679,32.418,-48.867,-179.852,6.155,149.066
C09890=1158.683,32.169,-48.852,-179.855,6.155,149.066
C09891=1158.689,31.919,-48.837,-179.857,6.153,149.067
C09892=1158.694,31.669,-48.822,-179.860,6.152,149.068
C09893=1158.699,31.420,-48.808,-179.862,6.152,149.068
C09894=1158.704,31.170,-48.792,-179.865,6.150,149.069
C09895=1158.709,30.921,-48.778,-179.868,6.149,149.069
C09896=1158.714,30.672,-48.763,-179.870,6.149,149.070
C09897=1158.719,30.422,-48.749,-179.872,6.148,149.070
C09898=1158.724,30.172,-48.734,-179.876,6.147,149.071
C09899=1158.729,29.923,-48.719,-179.878,6.146,149.071
C09900=1158.734,29.673,-48.705,-179.880,6.146,149.072
C09901=1158.739,29.424,-48.689,-179.883,6.144,149.073
C09902=1158.745,29.175,-48.675,-179.886,6.143,149.073
C09903=1158.750,28.925,-48.661,-179.888,6.143,149.074
C09904=1158.754,28.676,-48.646,-179.891,6.142,149.074
C09905=1158.760,28.426,-48.631,-179.893,6.140,149.075
C09906=1158.765,28.157,-48.615,-179.896,6.140,149.075
C09907=1158.770,27.888,-48.600,-179.899,6.138,149.076
C09908=1158.776,27.619,-48.584,-179.901,6.138,149.077
C09909=1158.781,27.350,-48.568,-179.904,6.137,149.077
C09910=1158.786,27.101,-48.553,-179.907,6.136,149.078
C09911=1158.791,26.851,-48.539,-179.909,6.135,149.078
C09912=1158.796,26.602,-48.524,-179.912,6.134,149.079
C09913=1158.802,26.352,-48.509,-179.914,6.134,149.080
C09914=1158.807,26.102,-48.495,-179.917,6.132,149.080
C09915=1158.812,25.853,-48.481,-179.920,6.132,149.081
C09916=1158.817,25.604,-48.466,-179.922,6.131,149.081
C09917=1158.822,25.354,-48.452,-179.924,6.131,149.082
C09918=1158.827,25.105,-48.437,-179.927,6.129,149.082
C09919=1158.832,24.855,-48.423,-179.930,6.128,149.083
C09920=1158.837,24.605,-48.408,-179.932,6.128,149.083
C09921=1158.842,24.356,-48.393,-179.935,6.127,149.084
C09922=1158.847,24.106,-48.379,-179.937,6.126,149.085
C09923=1158.853,23.857,-48.365,-179.940,6.125,149.085
C09924=1158.857,23.608,-48.350,-179.943,6.125,149.086
C09925=1158.862,23.358,-48.336,-179.945,6.124,149.086
C09926=1158.867,23.109,-48.322,-179.948,6.123,149.087
C09927=1158.873,22.858,-48.307,-179.950,6.122,149.087
C09928=1158.878,22.609,-48.292,-179.953,6.121,149.088
C09929=1158.883,22.359,-48.278,-179.955,6.120,149.089
C09930=1158.888,22.111,-48.264,-179.958,6.119,149.089
C09931=1158.893,21.861,-48.249,-179.961,6.118,149.090
C09932=1158.898,21.611,-48.235,-179.963,6.118,149.090
C09933=1158.903,21.362,-48.221,-179.965,6.117,149.091
C09934=1158.908,21.112,-48.206,-179.969,6.116,149.092
C09935=1158.913,20.862,-48.192,-179.971,6.115,149.092
C09936=1158.918,20.613,-48.178,-179.973,6.114,149.093
C09937=1158.923,20.363,-48.164,-179.976,6.114,149.093
C09938=1158.928,20.114,-48.150,-179.978,6.113,149.094
C09939=1158.933,19.864,-48.135,-179.981,6.111,149.094
C09940=1158.938,19.615,-48.120,-179.984,6.111,149.095
C09941=1158.943,19.366,-48.106,-179.986,6.110,149.095
C09942=1158.948,19.116,-48.092,-179.988,6.110,149.096
C09943=1158.953,18.866,-48.078,-179.991,6.108,149.097
C09944=1158.958,18.617,-48.064,-179.994,6.108,149.097
C09945=1158.963,18.367,-48.049,-179.996,6.107,149.098
C09946=1158.969,18.118,-48.035,-179.999,6.106,149.098
C09947=1158.974,17.868,-48.021,179.999,6.105,149.099
C09948=1158.979,17.619,-48.007,179.996,6.104,149.100
C09949=1158.984,17.369,-47.993,179.994,6.103,149.100
C09950=1158.989,17.120,-47.979,179.991,6.103,149.101
C09951=1158.994,16.870,-47.964,179.989,6.102,149.101
C09952=1158.999,16.620,-47.951,179.986,6.102,149.102
C09953=1159.004,16.370,-47.937,179.984,6.100,149.102
C09954=1159.010,16.121,-47.923,179.981,6.100,149.103
C09955=1159.015,15.871,-47.908,179.978,6.099,149.104
C09956=1159.020,15.622,-47.894,179.976,6.098,149.104
C09957=1159.025,15.372,-47.880,179.973,6.098,149.105
C09958=1159.030,15.123,-47.866,179.971,6.096,149.105
C09959=1159.035,14.873,-47.852,179.968,6.096,149.106
C09960=1159.039,14.624,-47.838,179.966,6.095,149.106
C09961=1159.045,14.375,-47.824,179.963,6.094,149.107
C09962=1159.050,14.125,-47.810,179.961,6.094,149.107
C09963=1159.055,13.875,-47.796,179.958,6.093,149.108
C09964=1159.060,13.625,-47.782,179.956,6.091,149.109
C09965=1159.066,13.376,-47.768,179.953,6.091,149.109
C09966=1159.071,13.126,-47.754,179.951,6.090,149.110
C09967=1159.076,12.877,-47.740,179.948,6.090,149.110
C09968=1159.080,12.628,-47.726,179.946,6.089,149.111
C09969=1159.086,12.378,-47.713,179.943,6.088,149.112
C09970=1159.091,12.128,-47.698,179.941,6.087,149.112
C09971=1159.096,11.879,-47.684,179.938,6.086,149.113
C09972=1159.101,11.629,-47.670,179.936,6.085,149.113
C09973=1159.106,11.379,-47.657,179.933,6.085,149.114
C09974=1159.111,11.130,-47.643,179.930,6.085,149.115
C09975=1159.116,10.880,-47.629,179.928,6.083,149.115
C09976=1159.121,10.631,-47.615,179.925,6.083,149.116
C09977=1159.127,10.381,-47.602,179.923,6.082,149.116
C09978=1159.132,10.131,-47.587,179.920,6.081,149.117
C09979=1159.136,9.882,-47.574,179.918,6.080,149.117
C09980=1159.142,9.633,-47.560,179.915,6.080,149.118
C09981=1159.147,9.383,-47.546,179.913,6.079,149.118
C09982=1159.153,9.134,-47.532,179.910,6.078,149.119
C09983=1159.158,8.884,-47.518,179.908,6.077,149.120
C09984=1159.162,8.634,-47.505,179.905,6.077,149.120
C09985=1159.168,8.385,-47.491,179.903,6.076,149.121
C09986=1159.173,8.135,-47.477,179.900,6.075,149.121
C09987=1159.178,7.886,-47.464,179.898,6.074,149.122
C09988=1159.183,7.636,-47.450,179.895,6.074,149.123
C09989=1159.188,7.386,-47.436,179.893,6.072,149.123
C09990=1159.193,7.137,-47.422,179.890,6.072,149.124
C09991=1159.198,6.887,-47.409,179.887,6.071,149.124
C09992=1159.204,6.638,-47.396,179.885,6.071,149.125
C09993=1159.209,6.388,-47.381,179.883,6.070,149.126
C09994=1159.213,6.139,-47.368,179.880,6.069,149.126
C09995=1159.219,5.889,-47.354,179.878,6.069,149.127
C09996=1159.224,5.639,-47.340,179.875,6.067,149.127
//INST
///DATE 2021/06/15 17:26
///ATTR SC,RW,RJ
////FRAME ROBOT
///GROUP1 RB1
NOP
MOVL C00000 V=800.0 PL=0
MOVL C00001 V=800.0 PL=0
MOVL C00002 V=800.0 PL=0
MOVL C00003 V=800.0 PL=0
MOVL C00004 V=800.0 PL=0
MOVL C00005 V=800.0 PL=0
MOVL C00006 V=800.0 PL=0
MOVL C00007 V=800.0 PL=0
MOVL C00008 V=800.0 PL=0
MOVL C00009 V=800.0 PL=0
MOVL C00010 V=800.0 PL=0
MOVL C00011 V=800.0 PL=0
MOVL C00012 V=800.0 PL=0
MOVL C00013 V=800.0 PL=0
MOVL C00014 V=800.0 PL=0
MOVL C00015 V=800.0 PL=0
MOVL C00016 V=800.0 PL=0
MOVL C00017 V=800.0 PL=0
MOVL C00018 V=800.0 PL=0
MOVL C00019 V=800.0 PL=0
MOVL C00020 V=800.0 PL=0
MOVL C00021 V=800.0 PL=0
MOVL C00022 V=800.0 PL=0
MOVL C00023 V=800.0 PL=0
MOVL C00024 V=800.0 PL=0
MOVL C00025 V=800.0 PL=0
MOVL C00026 V=800.0 PL=0
MOVL C00027 V=800.0 PL=0
MOVL C00028 V=800.0 PL=0
MOVL C00029 V=800.0 PL=0
MOVL C00030 V=800.0 PL=0
MOVL C00031 V=800.0 PL=0
MOVL C00032 V=800.0 PL=0
MOVL C00033 V=800.0 PL=0
MOVL C00034 V=800.0 PL=0
MOVL C00035 V=800.0 PL=0
MOVL C00036 V=800.0 PL=0
MOVL C00037 V=800.0 PL=0
MOVL C00038 V=800.0 PL=0
MOVL C00039 V=800.0 PL=0
MOVL C00040 V=800.0 PL=0
MOVL C00041 V=800.0 PL=0
MOVL C00042 V=800.0 PL=0
MOVL C00043 V=800.0 PL=0
MOVL C00044 V=800.0 PL=0
MOVL C00045 V=800.0 PL=0
MOVL C00046 V=800.0 PL=0
MOVL C00047 V=800.0 PL=0
MOVL C00048 V=800.0 PL=0
MOVL C00049 V=800.0 PL=0
MOVL C00050 V=800.0 PL=0
MOVL C00051 V=800.0 PL=0
MOVL C00052 V=800.0 PL=0
MOVL C00053 V=800.0 PL=0
MOVL C00054 V=800.0 PL=0
MOVL C00055 V=800.0 PL=0
MOVL C00056 V=800.0 PL=0
MOVL C00057 V=800.0 PL=0
MOVL C00058 V=800.0 PL=0
MOVL C00059 V=800.0 PL=0
MOVL C00060 V=800.0 PL=0
MOVL C00061 V=800.0 PL=0
MOVL C00062 V=800.0 PL=0
MOVL C00063 V=800.0 PL=0
MOVL C00064 V=800.0 PL=0
MOVL C00065 V=800.0 PL=0
MOVL C00066 V=800.0 PL=0
MOVL C00067 V=800.0 PL=0
MOVL C00068 V=800.0 PL=0
MOVL C00069 V=800.0 PL=0
MOVL C00070 V=800.0 PL=0
MOVL C00071 V=800.0 PL=0
MOVL C00072 V=800.0 PL=0
MOVL C00073 V=800.0 PL=0
MOVL C00074 V=800.0 PL=0
MOVL C00075 V=800.0 PL=0
MOVL C00076 V=800.0 PL=0
MOVL C00077 V=800.0 PL=0
MOVL C00078 V=800.0 PL=0
MOVL C00079 V=800.0 PL=0
MOVL C00080 V=800.0 PL=0
MOVL C00081 V=800.0 PL=0
MOVL C00082 V=800.0 PL=0
MOVL C00083 V=800.0 PL=0
MOVL C00084 V=800.0 PL=0
MOVL C00085 V=800.0 PL=0
MOVL C00086 V=800.0 PL=0
MOVL C00087 V=800.0 PL=0
MOVL C00088 V=800.0 PL=0
MOVL C00089 V=800.0 PL=0
MOVL C00090 V=800.0 PL=0
MOVL C00091 V=800.0 PL=0
MOVL C00092 V=800.0 PL=0
MOVL C00093 V=800.0 PL=0
MOVL C00094 V=800.0 PL=0
MOVL C00095 V=800.0 PL=0
MOVL C00096 V=800.0 PL=0
MOVL C00097 V=800.0 PL=0
MOVL C00098 V=800.0 PL=0
MOVL C00099 V=800.0 PL=0
MOVL C00100 V=800.0 PL=0
MOVL C00101 V=800.0 PL=0
MOVL C00102 V=800.0 PL=0
MOVL C00103 V=800.0 PL=0
MOVL C00104 V=800.0 PL=0
MOVL C00105 V=800.0 PL=0
MOVL C00106 V=800.0 PL=0
MOVL C00107 V=800.0 PL=0
MOVL C00108 V=800.0 PL=0
MOVL C00109 V=800.0 PL=0
MOVL C00110 V=800.0 PL=0
MOVL C00111 V=800.0 PL=0
MOVL C00112 V=800.0 PL=0
MOVL C00113 V=800.0 PL=0
MOVL C00114 V=800.0 PL=0
MOVL C00115 V=800.0 PL=0
MOVL C00116 V=800.0 PL=0
MOVL C00117 V=800.0 PL=0
MOVL C00118 V=800.0 PL=0
MOVL C00119 V=800.0 PL=0
MOVL C00120 V=800.0 PL=0
MOVL C00121 V=800.0 PL=0
MOVL C00122 V=800.0 PL=0
MOVL C00123 V=800.0 PL=0
MOVL C00124 V=800.0 PL=0
MOVL C00125 V=800.0 PL=0
MOVL C00126 V=800.0 PL=0
MOVL C00127 V=800.0 PL=0
MOVL C00128 V=800.0 PL=0
MOVL C00129 V=800.0 PL=0
MOVL C00130 V=800.0 PL=0
MOVL C00131 V=800.0 PL=0
MOVL C00132 V=800.0 PL=0
MOVL C00133 V=800.0 PL=0
MOVL C00134 V=800.0 PL=0
MOVL C00135 V=800.0 PL=0
MOVL C00136 V=800.0 PL=0
MOVL C00137 V=800.0 PL=0
MOVL C00138 V=800.0 PL=0
MOVL C00139 V=800.0 PL=0
MOVL C00140 V=800.0 PL=0
MOVL C00141 V=800.0 PL=0
MOVL C00142 V=800.0 PL=0
MOVL C00143 V=800.0 PL=0
MOVL C00144 V=800.0 PL=0
MOVL C00145 V=800.0 PL=0
MOVL C00146 V=800.0 PL=0
MOVL C00147 V=800.0 PL=0
MOVL C00148 V=800.0 PL=0
MOVL C00149 V=800.0 PL=0
MOVL C00150 V=800.0 PL=0
MOVL C00151 V=800.0 PL=0
MOVL C00152 V=800.0 PL=0
MOVL C00153 V=800.0 PL=0
MOVL C00154 V=800.0 PL=0
MOVL C00155 V=800.0 PL=0
MOVL C00156 V=800.0 PL=0
MOVL C00157 V=800.0 PL=0
MOVL C00158 V=800.0 PL=0
MOVL C00159 V=800.0 PL=0
MOVL C00160 V=800.0 PL=0
MOVL C00161 V=800.0 PL=0
MOVL C00162 V=800.0 PL=0
MOVL C00163 V=800.0 PL=0
MOVL C00164 V=800.0 PL=0
MOVL C00165 V=800.0 PL=0
MOVL C00166 V=800.0 PL=0
MOVL C00167 V=800.0 PL=0
MOVL C00168 V=800.0 PL=0
MOVL C00169 V=800.0 PL=0
MOVL C00170 V=800.0 PL=0
MOVL C00171 V=800.0 PL=0
MOVL C00172 V=800.0 PL=0
MOVL C00173 V=800.0 PL=0
MOVL C00174 V=800.0 PL=0
MOVL C00175 V=800.0 PL=0
MOVL C00176 V=800.0 PL=0
MOVL C00177 V=800.0 PL=0
MOVL C00178 V=800.0 PL=0
MOVL C00179 V=800.0 PL=0
MOVL C00180 V=800.0 PL=0
MOVL C00181 V=800.0 PL=0
MOVL C00182 V=800.0 PL=0
MOVL C00183 V=800.0 PL=0
MOVL C00184 V=800.0 PL=0
MOVL C00185 V=800.0 PL=0
MOVL C00186 V=800.0 PL=0
MOVL C00187 V=800.0 PL=0
MOVL C00188 V=800.0 PL=0
MOVL C00189 V=800.0 PL=0
MOVL C00190 V=800.0 PL=0
MOVL C00191 V=800.0 PL=0
MOVL C00192 V=800.0 PL=0
MOVL C00193 V=800.0 PL=0
MOVL C00194 V=800.0 PL=0
MOVL C00195 V=800.0 PL=0
MOVL C00196 V=800.0 PL=0
MOVL C00197 V=800.0 PL=0
MOVL C00198 V=800.0 PL=0
MOVL C00199 V=800.0 PL=0
MOVL C00200 V=800.0 PL=0
MOVL C00201 V=800.0 PL=0
MOVL C00202 V=800.0 PL=0
MOVL C00203 V=800.0 PL=0
MOVL C00204 V=800.0 PL=0
MOVL C00205 V=800.0 PL=0
MOVL C00206 V=800.0 PL=0
MOVL C00207 V=800.0 PL=0
MOVL C00208 V=800.0 PL=0
MOVL C00209 V=800.0 PL=0
MOVL C00210 V=800.0 PL=0
MOVL C00211 V=800.0 PL=0
MOVL C00212 V=800.0 PL=0
MOVL C00213 V=800.0 PL=0
MOVL C00214 V=800.0 PL=0
MOVL C00215 V=800.0 PL=0
MOVL C00216 V=800.0 PL=0
MOVL C00217 V=800.0 PL=0
MOVL C00218 V=800.0 PL=0
MOVL C00219 V=800.0 PL=0
MOVL C00220 V=800.0 PL=0
MOVL C00221 V=800.0 PL=0
MOVL C00222 V=800.0 PL=0
MOVL C00223 V=800.0 PL=0
MOVL C00224 V=800.0 PL=0
MOVL C00225 V=800.0 PL=0
MOVL C00226 V=800.0 PL=0
MOVL C00227 V=800.0 PL=0
MOVL C00228 V=800.0 PL=0
MOVL C00229 V=800.0 PL=0
MOVL C00230 V=800.0 PL=0
MOVL C00231 V=800.0 PL=0
MOVL C00232 V=800.0 PL=0
MOVL C00233 V=800.0 PL=0
MOVL C00234 V=800.0 PL=0
MOVL C00235 V=800.0 PL=0
MOVL C00236 V=800.0 PL=0
MOVL C00237 V=800.0 PL=0
MOVL C00238 V=800.0 PL=0
MOVL C00239 V=800.0 PL=0
MOVL C00240 V=800.0 PL=0
MOVL C00241 V=800.0 PL=0
MOVL C00242 V=800.0 PL=0
MOVL C00243 V=800.0 PL=0
MOVL C00244 V=800.0 PL=0
MOVL C00245 V=800.0 PL=0
MOVL C00246 V=800.0 PL=0
MOVL C00247 V=800.0 PL=0
MOVL C00248 V=800.0 PL=0
MOVL C00249 V=800.0 PL=0
MOVL C00250 V=800.0 PL=0
MOVL C00251 V=800.0 PL=0
MOVL C00252 V=800.0 PL=0
MOVL C00253 V=800.0 PL=0
MOVL C00254 V=800.0 PL=0
MOVL C00255 V=800.0 PL=0
MOVL C00256 V=800.0 PL=0
MOVL C00257 V=800.0 PL=0
MOVL C00258 V=800.0 PL=0
MOVL C00259 V=800.0 PL=0
MOVL C00260 V=800.0 PL=0
MOVL C00261 V=800.0 PL=0
MOVL C00262 V=800.0 PL=0
MOVL C00263 V=800.0 PL=0
MOVL C00264 V=800.0 PL=0
MOVL C00265 V=800.0 PL=0
MOVL C00266 V=800.0 PL=0
MOVL C00267 V=800.0 PL=0
MOVL C00268 V=800.0 PL=0
MOVL C00269 V=800.0 PL=0
MOVL C00270 V=800.0 PL=0
MOVL C00271 V=800.0 PL=0
MOVL C00272 V=800.0 PL=0
MOVL C00273 V=800.0 PL=0
MOVL C00274 V=800.0 PL=0
MOVL C00275 V=800.0 PL=0
MOVL C00276 V=800.0 PL=0
MOVL C00277 V=800.0 PL=0
MOVL C00278 V=800.0 PL=0
MOVL C00279 V=800.0 PL=0
MOVL C00280 V=800.0 PL=0
MOVL C00281 V=800.0 PL=0
MOVL C00282 V=800.0 PL=0
MOVL C00283 V=800.0 PL=0
MOVL C00284 V=800.0 PL=0
MOVL C00285 V=800.0 PL=0
MOVL C00286 V=800.0 PL=0
MOVL C00287 V=800.0 PL=0
MOVL C00288 V=800.0 PL=0
MOVL C00289 V=800.0 PL=0
MOVL C00290 V=800.0 PL=0
MOVL C00291 V=800.0 PL=0
MOVL C00292 V=800.0 PL=0
MOVL C00293 V=800.0 PL=0
MOVL C00294 V=800.0 PL=0
MOVL C00295 V=800.0 PL=0
MOVL C00296 V=800.0 PL=0
MOVL C00297 V=800.0 PL=0
MOVL C00298 V=800.0 PL=0
MOVL C00299 V=800.0 PL=0
MOVL C00300 V=800.0 PL=0
MOVL C00301 V=800.0 PL=0
MOVL C00302 V=800.0 PL=0
MOVL C00303 V=800.0 PL=0
MOVL C00304 V=800.0 PL=0
MOVL C00305 V=800.0 PL=0
MOVL C00306 V=800.0 PL=0
MOVL C00307 V=800.0 PL=0
MOVL C00308 V=800.0 PL=0
MOVL C00309 V=800.0 PL=0
MOVL C00310 V=800.0 PL=0
MOVL C00311 V=800.0 PL=0
MOVL C00312 V=800.0 PL=0
MOVL C00313 V=800.0 PL=0
MOVL C00314 V=800.0 PL=0
MOVL C00315 V=800.0 PL=0
MOVL C00316 V=800.0 PL=0
MOVL C00317 V=800.0 PL=0
MOVL C00318 V=800.0 PL=0
MOVL C00319 V=800.0 PL=0
MOVL C00320 V=800.0 PL=0
MOVL C00321 V=800.0 PL=0
MOVL C00322 V=800.0 PL=0
MOVL C00323 V=800.0 PL=0
MOVL C00324 V=800.0 PL=0
MOVL C00325 V=800.0 PL=0
MOVL C00326 V=800.0 PL=0
MOVL C00327 V=800.0 PL=0
MOVL C00328 V=800.0 PL=0
MOVL C00329 V=800.0 PL=0
MOVL C00330 V=800.0 PL=0
MOVL C00331 V=800.0 PL=0
MOVL C00332 V=800.0 PL=0
MOVL C00333 V=800.0 PL=0
MOVL C00334 V=800.0 PL=0
MOVL C00335 V=800.0 PL=0
MOVL C00336 V=800.0 PL=0
MOVL C00337 V=800.0 PL=0
MOVL C00338 V=800.0 PL=0
MOVL C00339 V=800.0 PL=0
MOVL C00340 V=800.0 PL=0
MOVL C00341 V=800.0 PL=0
MOVL C00342 V=800.0 PL=0
MOVL C00343 V=800.0 PL=0
MOVL C00344 V=800.0 PL=0
MOVL C00345 V=800.0 PL=0
MOVL C00346 V=800.0 PL=0
MOVL C00347 V=800.0 PL=0
MOVL C00348 V=800.0 PL=0
MOVL C00349 V=800.0 PL=0
MOVL C00350 V=800.0 PL=0
MOVL C00351 V=800.0 PL=0
MOVL C00352 V=800.0 PL=0
MOVL C00353 V=800.0 PL=0
MOVL C00354 V=800.0 PL=0
MOVL C00355 V=800.0 PL=0
MOVL C00356 V=800.0 PL=0
MOVL C00357 V=800.0 PL=0
MOVL C00358 V=800.0 PL=0
MOVL C00359 V=800.0 PL=0
MOVL C00360 V=800.0 PL=0
MOVL C00361 V=800.0 PL=0
MOVL C00362 V=800.0 PL=0
MOVL C00363 V=800.0 PL=0
MOVL C00364 V=800.0 PL=0
MOVL C00365 V=800.0 PL=0
MOVL C00366 V=800.0 PL=0
MOVL C00367 V=800.0 PL=0
MOVL C00368 V=800.0 PL=0
MOVL C00369 V=800.0 PL=0
MOVL C00370 V=800.0 PL=0
MOVL C00371 V=800.0 PL=0
MOVL C00372 V=800.0 PL=0
MOVL C00373 V=800.0 PL=0
MOVL C00374 V=800.0 PL=0
MOVL C00375 V=800.0 PL=0
MOVL C00376 V=800.0 PL=0
MOVL C00377 V=800.0 PL=0
MOVL C00378 V=800.0 PL=0
MOVL C00379 V=800.0 PL=0
MOVL C00380 V=800.0 PL=0
MOVL C00381 V=800.0 PL=0
MOVL C00382 V=800.0 PL=0
MOVL C00383 V=800.0 PL=0
MOVL C00384 V=800.0 PL=0
MOVL C00385 V=800.0 PL=0
MOVL C00386 V=800.0 PL=0
MOVL C00387 V=800.0 PL=0
MOVL C00388 V=800.0 PL=0
MOVL C00389 V=800.0 PL=0
MOVL C00390 V=800.0 PL=0
MOVL C00391 V=800.0 PL=0
MOVL C00392 V=800.0 PL=0
MOVL C00393 V=800.0 PL=0
MOVL C00394 V=800.0 PL=0
MOVL C00395 V=800.0 PL=0
MOVL C00396 V=800.0 PL=0
MOVL C00397 V=800.0 PL=0
MOVL C00398 V=800.0 PL=0
MOVL C00399 V=800.0 PL=0
MOVL C00400 V=800.0 PL=0
MOVL C00401 V=800.0 PL=0
MOVL C00402 V=800.0 PL=0
MOVL C00403 V=800.0 PL=0
MOVL C00404 V=800.0 PL=0
MOVL C00405 V=800.0 PL=0
MOVL C00406 V=800.0 PL=0
MOVL C00407 V=800.0 PL=0
MOVL C00408 V=800.0 PL=0
MOVL C00409 V=800.0 PL=0
MOVL C00410 V=800.0 PL=0
MOVL C00411 V=800.0 PL=0
MOVL C00412 V=800.0 PL=0
MOVL C00413 V=800.0 PL=0
MOVL C00414 V=800.0 PL=0
MOVL C00415 V=800.0 PL=0
MOVL C00416 V=800.0 PL=0
MOVL C00417 V=800.0 PL=0
MOVL C00418 V=800.0 PL=0
MOVL C00419 V=800.0 PL=0
MOVL C00420 V=800.0 PL=0
MOVL C00421 V=800.0 PL=0
MOVL C00422 V=800.0 PL=0
MOVL C00423 V=800.0 PL=0
MOVL C00424 V=800.0 PL=0
MOVL C00425 V=800.0 PL=0
MOVL C00426 V=800.0 PL=0
MOVL C00427 V=800.0 PL=0
MOVL C00428 V=800.0 PL=0
MOVL C00429 V=800.0 PL=0
MOVL C00430 V=800.0 PL=0
MOVL C00431 V=800.0 PL=0
MOVL C00432 V=800.0 PL=0
MOVL C00433 V=800.0 PL=0
MOVL C00434 V=800.0 PL=0
MOVL C00435 V=800.0 PL=0
MOVL C00436 V=800.0 PL=0
MOVL C00437 V=800.0 PL=0
MOVL C00438 V=800.0 PL=0
MOVL C00439 V=800.0 PL=0
MOVL C00440 V=800.0 PL=0
MOVL C00441 V=800.0 PL=0
MOVL C00442 V=800.0 PL=0
MOVL C00443 V=800.0 PL=0
MOVL C00444 V=800.0 PL=0
MOVL C00445 V=800.0 PL=0
MOVL C00446 V=800.0 PL=0
MOVL C00447 V=800.0 PL=0
MOVL C00448 V=800.0 PL=0
MOVL C00449 V=800.0 PL=0
MOVL C00450 V=800.0 PL=0
MOVL C00451 V=800.0 PL=0
MOVL C00452 V=800.0 PL=0
MOVL C00453 V=800.0 PL=0
MOVL C00454 V=800.0 PL=0
MOVL C00455 V=800.0 PL=0
MOVL C00456 V=800.0 PL=0
MOVL C00457 V=800.0 PL=0
MOVL C00458 V=800.0 PL=0
MOVL C00459 V=800.0 PL=0
MOVL C00460 V=800.0 PL=0
MOVL C00461 V=800.0 PL=0
MOVL C00462 V=800.0 PL=0
MOVL C00463 V=800.0 PL=0
MOVL C00464 V=800.0 PL=0
MOVL C00465 V=800.0 PL=0
MOVL C00466 V=800.0 PL=0
MOVL C00467 V=800.0 PL=0
MOVL C00468 V=800.0 PL=0
MOVL C00469 V=800.0 PL=0
MOVL C00470 V=800.0 PL=0
MOVL C00471 V=800.0 PL=0
MOVL C00472 V=800.0 PL=0
MOVL C00473 V=800.0 PL=0
MOVL C00474 V=800.0 PL=0
MOVL C00475 V=800.0 PL=0
MOVL C00476 V=800.0 PL=0
MOVL C00477 V=800.0 PL=0
MOVL C00478 V=800.0 PL=0
MOVL C00479 V=800.0 PL=0
MOVL C00480 V=800.0 PL=0
MOVL C00481 V=800.0 PL=0
MOVL C00482 V=800.0 PL=0
MOVL C00483 V=800.0 PL=0
MOVL C00484 V=800.0 PL=0
MOVL C00485 V=800.0 PL=0
MOVL C00486 V=800.0 PL=0
MOVL C00487 V=800.0 PL=0
MOVL C00488 V=800.0 PL=0
MOVL C00489 V=800.0 PL=0
MOVL C00490 V=800.0 PL=0
MOVL C00491 V=800.0 PL=0
MOVL C00492 V=800.0 PL=0
MOVL C00493 V=800.0 PL=0
MOVL C00494 V=800.0 PL=0
MOVL C00495 V=800.0 PL=0
MOVL C00496 V=800.0 PL=0
MOVL C00497 V=800.0 PL=0
MOVL C00498 V=800.0 PL=0
MOVL C00499 V=800.0 PL=0
MOVL C00500 V=800.0 PL=0
MOVL C00501 V=800.0 PL=0
MOVL C00502 V=800.0 PL=0
MOVL C00503 V=800.0 PL=0
MOVL C00504 V=800.0 PL=0
MOVL C00505 V=800.0 PL=0
MOVL C00506 V=800.0 PL=0
MOVL C00507 V=800.0 PL=0
MOVL C00508 V=800.0 PL=0
MOVL C00509 V=800.0 PL=0
MOVL C00510 V=800.0 PL=0
MOVL C00511 V=800.0 PL=0
MOVL C00512 V=800.0 PL=0
MOVL C00513 V=800.0 PL=0
MOVL C00514 V=800.0 PL=0
MOVL C00515 V=800.0 PL=0
MOVL C00516 V=800.0 PL=0
MOVL C00517 V=800.0 PL=0
MOVL C00518 V=800.0 PL=0
MOVL C00519 V=800.0 PL=0
MOVL C00520 V=800.0 PL=0
MOVL C00521 V=800.0 PL=0
MOVL C00522 V=800.0 PL=0
MOVL C00523 V=800.0 PL=0
MOVL C00524 V=800.0 PL=0
MOVL C00525 V=800.0 PL=0
MOVL C00526 V=800.0 PL=0
MOVL C00527 V=800.0 PL=0
MOVL C00528 V=800.0 PL=0
MOVL C00529 V=800.0 PL=0
MOVL C00530 V=800.0 PL=0
MOVL C00531 V=800.0 PL=0
MOVL C00532 V=800.0 PL=0
MOVL C00533 V=800.0 PL=0
MOVL C00534 V=800.0 PL=0
MOVL C00535 V=800.0 PL=0
MOVL C00536 V=800.0 PL=0
MOVL C00537 V=800.0 PL=0
MOVL C00538 V=800.0 PL=0
MOVL C00539 V=800.0 PL=0
MOVL C00540 V=800.0 PL=0
MOVL C00541 V=800.0 PL=0
MOVL C00542 V=800.0 PL=0
MOVL C00543 V=800.0 PL=0
MOVL C00544 V=800.0 PL=0
MOVL C00545 V=800.0 PL=0
MOVL C00546 V=800.0 PL=0
MOVL C00547 V=800.0 PL=0
MOVL C00548 V=800.0 PL=0
MOVL C00549 V=800.0 PL=0
MOVL C00550 V=800.0 PL=0
MOVL C00551 V=800.0 PL=0
MOVL C00552 V=800.0 PL=0
MOVL C00553 V=800.0 PL=0
MOVL C00554 V=800.0 PL=0
MOVL C00555 V=800.0 PL=0
MOVL C00556 V=800.0 PL=0
MOVL C00557 V=800.0 PL=0
MOVL C00558 V=800.0 PL=0
MOVL C00559 V=800.0 PL=0
MOVL C00560 V=800.0 PL=0
MOVL C00561 V=800.0 PL=0
MOVL C00562 V=800.0 PL=0
MOVL C00563 V=800.0 PL=0
MOVL C00564 V=800.0 PL=0
MOVL C00565 V=800.0 PL=0
MOVL C00566 V=800.0 PL=0
MOVL C00567 V=800.0 PL=0
MOVL C00568 V=800.0 PL=0
MOVL C00569 V=800.0 PL=0
MOVL C00570 V=800.0 PL=0
MOVL C00571 V=800.0 PL=0
MOVL C00572 V=800.0 PL=0
MOVL C00573 V=800.0 PL=0
MOVL C00574 V=800.0 PL=0
MOVL C00575 V=800.0 PL=0
MOVL C00576 V=800.0 PL=0
MOVL C00577 V=800.0 PL=0
MOVL C00578 V=800.0 PL=0
MOVL C00579 V=800.0 PL=0
MOVL C00580 V=800.0 PL=0
MOVL C00581 V=800.0 PL=0
MOVL C00582 V=800.0 PL=0
MOVL C00583 V=800.0 PL=0
MOVL C00584 V=800.0 PL=0
MOVL C00585 V=800.0 PL=0
MOVL C00586 V=800.0 PL=0
MOVL C00587 V=800.0 PL=0
MOVL C00588 V=800.0 PL=0
MOVL C00589 V=800.0 PL=0
MOVL C00590 V=800.0 PL=0
MOVL C00591 V=800.0 PL=0
MOVL C00592 V=800.0 PL=0
MOVL C00593 V=800.0 PL=0
MOVL C00594 V=800.0 PL=0
MOVL C00595 V=800.0 PL=0
MOVL C00596 V=800.0 PL=0
MOVL C00597 V=800.0 PL=0
MOVL C00598 V=800.0 PL=0
MOVL C00599 V=800.0 PL=0
MOVL C00600 V=800.0 PL=0
MOVL C00601 V=800.0 PL=0
MOVL C00602 V=800.0 PL=0
MOVL C00603 V=800.0 PL=0
MOVL C00604 V=800.0 PL=0
MOVL C00605 V=800.0 PL=0
MOVL C00606 V=800.0 PL=0
MOVL C00607 V=800.0 PL=0
MOVL C00608 V=800.0 PL=0
MOVL C00609 V=800.0 PL=0
MOVL C00610 V=800.0 PL=0
MOVL C00611 V=800.0 PL=0
MOVL C00612 V=800.0 PL=0
MOVL C00613 V=800.0 PL=0
MOVL C00614 V=800.0 PL=0
MOVL C00615 V=800.0 PL=0
MOVL C00616 V=800.0 PL=0
MOVL C00617 V=800.0 PL=0
MOVL C00618 V=800.0 PL=0
MOVL C00619 V=800.0 PL=0
MOVL C00620 V=800.0 PL=0
MOVL C00621 V=800.0 PL=0
MOVL C00622 V=800.0 PL=0
MOVL C00623 V=800.0 PL=0
MOVL C00624 V=800.0 PL=0
MOVL C00625 V=800.0 PL=0
MOVL C00626 V=800.0 PL=0
MOVL C00627 V=800.0 PL=0
MOVL C00628 V=800.0 PL=0
MOVL C00629 V=800.0 PL=0
MOVL C00630 V=800.0 PL=0
MOVL C00631 V=800.0 PL=0
MOVL C00632 V=800.0 PL=0
MOVL C00633 V=800.0 PL=0
MOVL C00634 V=800.0 PL=0
MOVL C00635 V=800.0 PL=0
MOVL C00636 V=800.0 PL=0
MOVL C00637 V=800.0 PL=0
MOVL C00638 V=800.0 PL=0
MOVL C00639 V=800.0 PL=0
MOVL C00640 V=800.0 PL=0
MOVL C00641 V=800.0 PL=0
MOVL C00642 V=800.0 PL=0
MOVL C00643 V=800.0 PL=0
MOVL C00644 V=800.0 PL=0
MOVL C00645 V=800.0 PL=0
MOVL C00646 V=800.0 PL=0
MOVL C00647 V=800.0 PL=0
MOVL C00648 V=800.0 PL=0
MOVL C00649 V=800.0 PL=0
MOVL C00650 V=800.0 PL=0
MOVL C00651 V=800.0 PL=0
MOVL C00652 V=800.0 PL=0
MOVL C00653 V=800.0 PL=0
MOVL C00654 V=800.0 PL=0
MOVL C00655 V=800.0 PL=0
MOVL C00656 V=800.0 PL=0
MOVL C00657 V=800.0 PL=0
MOVL C00658 V=800.0 PL=0
MOVL C00659 V=800.0 PL=0
MOVL C00660 V=800.0 PL=0
MOVL C00661 V=800.0 PL=0
MOVL C00662 V=800.0 PL=0
MOVL C00663 V=800.0 PL=0
MOVL C00664 V=800.0 PL=0
MOVL C00665 V=800.0 PL=0
MOVL C00666 V=800.0 PL=0
MOVL C00667 V=800.0 PL=0
MOVL C00668 V=800.0 PL=0
MOVL C00669 V=800.0 PL=0
MOVL C00670 V=800.0 PL=0
MOVL C00671 V=800.0 PL=0
MOVL C00672 V=800.0 PL=0
MOVL C00673 V=800.0 PL=0
MOVL C00674 V=800.0 PL=0
MOVL C00675 V=800.0 PL=0
MOVL C00676 V=800.0 PL=0
MOVL C00677 V=800.0 PL=0
MOVL C00678 V=800.0 PL=0
MOVL C00679 V=800.0 PL=0
MOVL C00680 V=800.0 PL=0
MOVL C00681 V=800.0 PL=0
MOVL C00682 V=800.0 PL=0
MOVL C00683 V=800.0 PL=0
MOVL C00684 V=800.0 PL=0
MOVL C00685 V=800.0 PL=0
MOVL C00686 V=800.0 PL=0
MOVL C00687 V=800.0 PL=0
MOVL C00688 V=800.0 PL=0
MOVL C00689 V=800.0 PL=0
MOVL C00690 V=800.0 PL=0
MOVL C00691 V=800.0 PL=0
MOVL C00692 V=800.0 PL=0
MOVL C00693 V=800.0 PL=0
MOVL C00694 V=800.0 PL=0
MOVL C00695 V=800.0 PL=0
MOVL C00696 V=800.0 PL=0
MOVL C00697 V=800.0 PL=0
MOVL C00698 V=800.0 PL=0
MOVL C00699 V=800.0 PL=0
MOVL C00700 V=800.0 PL=0
MOVL C00701 V=800.0 PL=0
MOVL C00702 V=800.0 PL=0
MOVL C00703 V=800.0 PL=0
MOVL C00704 V=800.0 PL=0
MOVL C00705 V=800.0 PL=0
MOVL C00706 V=800.0 PL=0
MOVL C00707 V=800.0 PL=0
MOVL C00708 V=800.0 PL=0
MOVL C00709 V=800.0 PL=0
MOVL C00710 V=800.0 PL=0
MOVL C00711 V=800.0 PL=0
MOVL C00712 V=800.0 PL=0
MOVL C00713 V=800.0 PL=0
MOVL C00714 V=800.0 PL=0
MOVL C00715 V=800.0 PL=0
MOVL C00716 V=800.0 PL=0
MOVL C00717 V=800.0 PL=0
MOVL C00718 V=800.0 PL=0
MOVL C00719 V=800.0 PL=0
MOVL C00720 V=800.0 PL=0
MOVL C00721 V=800.0 PL=0
MOVL C00722 V=800.0 PL=0
MOVL C00723 V=800.0 PL=0
MOVL C00724 V=800.0 PL=0
MOVL C00725 V=800.0 PL=0
MOVL C00726 V=800.0 PL=0
MOVL C00727 V=800.0 PL=0
MOVL C00728 V=800.0 PL=0
MOVL C00729 V=800.0 PL=0
MOVL C00730 V=800.0 PL=0
MOVL C00731 V=800.0 PL=0
MOVL C00732 V=800.0 PL=0
MOVL C00733 V=800.0 PL=0
MOVL C00734 V=800.0 PL=0
MOVL C00735 V=800.0 PL=0
MOVL C00736 V=800.0 PL=0
MOVL C00737 V=800.0 PL=0
MOVL C00738 V=800.0 PL=0
MOVL C00739 V=800.0 PL=0
MOVL C00740 V=800.0 PL=0
MOVL C00741 V=800.0 PL=0
MOVL C00742 V=800.0 PL=0
MOVL C00743 V=800.0 PL=0
MOVL C00744 V=800.0 PL=0
MOVL C00745 V=800.0 PL=0
MOVL C00746 V=800.0 PL=0
MOVL C00747 V=800.0 PL=0
MOVL C00748 V=800.0 PL=0
MOVL C00749 V=800.0 PL=0
MOVL C00750 V=800.0 PL=0
MOVL C00751 V=800.0 PL=0
MOVL C00752 V=800.0 PL=0
MOVL C00753 V=800.0 PL=0
MOVL C00754 V=800.0 PL=0
MOVL C00755 V=800.0 PL=0
MOVL C00756 V=800.0 PL=0
MOVL C00757 V=800.0 PL=0
MOVL C00758 V=800.0 PL=0
MOVL C00759 V=800.0 PL=0
MOVL C00760 V=800.0 PL=0
MOVL C00761 V=800.0 PL=0
MOVL C00762 V=800.0 PL=0
MOVL C00763 V=800.0 PL=0
MOVL C00764 V=800.0 PL=0
MOVL C00765 V=800.0 PL=0
MOVL C00766 V=800.0 PL=0
MOVL C00767 V=800.0 PL=0
MOVL C00768 V=800.0 PL=0
MOVL C00769 V=800.0 PL=0
MOVL C00770 V=800.0 PL=0
MOVL C00771 V=800.0 PL=0
MOVL C00772 V=800.0 PL=0
MOVL C00773 V=800.0 PL=0
MOVL C00774 V=800.0 PL=0
MOVL C00775 V=800.0 PL=0
MOVL C00776 V=800.0 PL=0
MOVL C00777 V=800.0 PL=0
MOVL C00778 V=800.0 PL=0
MOVL C00779 V=800.0 PL=0
MOVL C00780 V=800.0 PL=0
MOVL C00781 V=800.0 PL=0
MOVL C00782 V=800.0 PL=0
MOVL C00783 V=800.0 PL=0
MOVL C00784 V=800.0 PL=0
MOVL C00785 V=800.0 PL=0
MOVL C00786 V=800.0 PL=0
MOVL C00787 V=800.0 PL=0
MOVL C00788 V=800.0 PL=0
MOVL C00789 V=800.0 PL=0
MOVL C00790 V=800.0 PL=0
MOVL C00791 V=800.0 PL=0
MOVL C00792 V=800.0 PL=0
MOVL C00793 V=800.0 PL=0
MOVL C00794 V=800.0 PL=0
MOVL C00795 V=800.0 PL=0
MOVL C00796 V=800.0 PL=0
MOVL C00797 V=800.0 PL=0
MOVL C00798 V=800.0 PL=0
MOVL C00799 V=800.0 PL=0
MOVL C00800 V=800.0 PL=0
MOVL C00801 V=800.0 PL=0
MOVL C00802 V=800.0 PL=0
MOVL C00803 V=800.0 PL=0
MOVL C00804 V=800.0 PL=0
MOVL C00805 V=800.0 PL=0
MOVL C00806 V=800.0 PL=0
MOVL C00807 V=800.0 PL=0
MOVL C00808 V=800.0 PL=0
MOVL C00809 V=800.0 PL=0
MOVL C00810 V=800.0 PL=0
MOVL C00811 V=800.0 PL=0
MOVL C00812 V=800.0 PL=0
MOVL C00813 V=800.0 PL=0
MOVL C00814 V=800.0 PL=0
MOVL C00815 V=800.0 PL=0
MOVL C00816 V=800.0 PL=0
MOVL C00817 V=800.0 PL=0
MOVL C00818 V=800.0 PL=0
MOVL C00819 V=800.0 PL=0
MOVL C00820 V=800.0 PL=0
MOVL C00821 V=800.0 PL=0
MOVL C00822 V=800.0 PL=0
MOVL C00823 V=800.0 PL=0
MOVL C00824 V=800.0 PL=0
MOVL C00825 V=800.0 PL=0
MOVL C00826 V=800.0 PL=0
MOVL C00827 V=800.0 PL=0
MOVL C00828 V=800.0 PL=0
MOVL C00829 V=800.0 PL=0
MOVL C00830 V=800.0 PL=0
MOVL C00831 V=800.0 PL=0
MOVL C00832 V=800.0 PL=0
MOVL C00833 V=800.0 PL=0
MOVL C00834 V=800.0 PL=0
MOVL C00835 V=800.0 PL=0
MOVL C00836 V=800.0 PL=0
MOVL C00837 V=800.0 PL=0
MOVL C00838 V=800.0 PL=0
MOVL C00839 V=800.0 PL=0
MOVL C00840 V=800.0 PL=0
MOVL C00841 V=800.0 PL=0
MOVL C00842 V=800.0 PL=0
MOVL C00843 V=800.0 PL=0
MOVL C00844 V=800.0 PL=0
MOVL C00845 V=800.0 PL=0
MOVL C00846 V=800.0 PL=0
MOVL C00847 V=800.0 PL=0
MOVL C00848 V=800.0 PL=0
MOVL C00849 V=800.0 PL=0
MOVL C00850 V=800.0 PL=0
MOVL C00851 V=800.0 PL=0
MOVL C00852 V=800.0 PL=0
MOVL C00853 V=800.0 PL=0
MOVL C00854 V=800.0 PL=0
MOVL C00855 V=800.0 PL=0
MOVL C00856 V=800.0 PL=0
MOVL C00857 V=800.0 PL=0
MOVL C00858 V=800.0 PL=0
MOVL C00859 V=800.0 PL=0
MOVL C00860 V=800.0 PL=0
MOVL C00861 V=800.0 PL=0
MOVL C00862 V=800.0 PL=0
MOVL C00863 V=800.0 PL=0
MOVL C00864 V=800.0 PL=0
MOVL C00865 V=800.0 PL=0
MOVL C00866 V=800.0 PL=0
MOVL C00867 V=800.0 PL=0
MOVL C00868 V=800.0 PL=0
MOVL C00869 V=800.0 PL=0
MOVL C00870 V=800.0 PL=0
MOVL C00871 V=800.0 PL=0
MOVL C00872 V=800.0 PL=0
MOVL C00873 V=800.0 PL=0
MOVL C00874 V=800.0 PL=0
MOVL C00875 V=800.0 PL=0
MOVL C00876 V=800.0 PL=0
MOVL C00877 V=800.0 PL=0
MOVL C00878 V=800.0 PL=0
MOVL C00879 V=800.0 PL=0
MOVL C00880 V=800.0 PL=0
MOVL C00881 V=800.0 PL=0
MOVL C00882 V=800.0 PL=0
MOVL C00883 V=800.0 PL=0
MOVL C00884 V=800.0 PL=0
MOVL C00885 V=800.0 PL=0
MOVL C00886 V=800.0 PL=0
MOVL C00887 V=800.0 PL=0
MOVL C00888 V=800.0 PL=0
MOVL C00889 V=800.0 PL=0
MOVL C00890 V=800.0 PL=0
MOVL C00891 V=800.0 PL=0
MOVL C00892 V=800.0 PL=0
MOVL C00893 V=800.0 PL=0
MOVL C00894 V=800.0 PL=0
MOVL C00895 V=800.0 PL=0
MOVL C00896 V=800.0 PL=0
MOVL C00897 V=800.0 PL=0
MOVL C00898 V=800.0 PL=0
MOVL C00899 V=800.0 PL=0
MOVL C00900 V=800.0 PL=0
MOVL C00901 V=800.0 PL=0
MOVL C00902 V=800.0 PL=0
MOVL C00903 V=800.0 PL=0
MOVL C00904 V=800.0 PL=0
MOVL C00905 V=800.0 PL=0
MOVL C00906 V=800.0 PL=0
MOVL C00907 V=800.0 PL=0
MOVL C00908 V=800.0 PL=0
MOVL C00909 V=800.0 PL=0
MOVL C00910 V=800.0 PL=0
MOVL C00911 V=800.0 PL=0
MOVL C00912 V=800.0 PL=0
MOVL C00913 V=800.0 PL=0
MOVL C00914 V=800.0 PL=0
MOVL C00915 V=800.0 PL=0
MOVL C00916 V=800.0 PL=0
MOVL C00917 V=800.0 PL=0
MOVL C00918 V=800.0 PL=0
MOVL C00919 V=800.0 PL=0
MOVL C00920 V=800.0 PL=0
MOVL C00921 V=800.0 PL=0
MOVL C00922 V=800.0 PL=0
MOVL C00923 V=800.0 PL=0
MOVL C00924 V=800.0 PL=0
MOVL C00925 V=800.0 PL=0
MOVL C00926 V=800.0 PL=0
MOVL C00927 V=800.0 PL=0
MOVL C00928 V=800.0 PL=0
MOVL C00929 V=800.0 PL=0
MOVL C00930 V=800.0 PL=0
MOVL C00931 V=800.0 PL=0
MOVL C00932 V=800.0 PL=0
MOVL C00933 V=800.0 PL=0
MOVL C00934 V=800.0 PL=0
MOVL C00935 V=800.0 PL=0
MOVL C00936 V=800.0 PL=0
MOVL C00937 V=800.0 PL=0
MOVL C00938 V=800.0 PL=0
MOVL C00939 V=800.0 PL=0
MOVL C00940 V=800.0 PL=0
MOVL C00941 V=800.0 PL=0
MOVL C00942 V=800.0 PL=0
MOVL C00943 V=800.0 PL=0
MOVL C00944 V=800.0 PL=0
MOVL C00945 V=800.0 PL=0
MOVL C00946 V=800.0 PL=0
MOVL C00947 V=800.0 PL=0
MOVL C00948 V=800.0 PL=0
MOVL C00949 V=800.0 PL=0
MOVL C00950 V=800.0 PL=0
MOVL C00951 V=800.0 PL=0
MOVL C00952 V=800.0 PL=0
MOVL C00953 V=800.0 PL=0
MOVL C00954 V=800.0 PL=0
MOVL C00955 V=800.0 PL=0
MOVL C00956 V=800.0 PL=0
MOVL C00957 V=800.0 PL=0
MOVL C00958 V=800.0 PL=0
MOVL C00959 V=800.0 PL=0
MOVL C00960 V=800.0 PL=0
MOVL C00961 V=800.0 PL=0
MOVL C00962 V=800.0 PL=0
MOVL C00963 V=800.0 PL=0
MOVL C00964 V=800.0 PL=0
MOVL C00965 V=800.0 PL=0
MOVL C00966 V=800.0 PL=0
MOVL C00967 V=800.0 PL=0
MOVL C00968 V=800.0 PL=0
MOVL C00969 V=800.0 PL=0
MOVL C00970 V=800.0 PL=0
MOVL C00971 V=800.0 PL=0
MOVL C00972 V=800.0 PL=0
MOVL C00973 V=800.0 PL=0
MOVL C00974 V=800.0 PL=0
MOVL C00975 V=800.0 PL=0
MOVL C00976 V=800.0 PL=0
MOVL C00977 V=800.0 PL=0
MOVL C00978 V=800.0 PL=0
MOVL C00979 V=800.0 PL=0
MOVL C00980 V=800.0 PL=0
MOVL C00981 V=800.0 PL=0
MOVL C00982 V=800.0 PL=0
MOVL C00983 V=800.0 PL=0
MOVL C00984 V=800.0 PL=0
MOVL C00985 V=800.0 PL=0
MOVL C00986 V=800.0 PL=0
MOVL C00987 V=800.0 PL=0
MOVL C00988 V=800.0 PL=0
MOVL C00989 V=800.0 PL=0
MOVL C00990 V=800.0 PL=0
MOVL C00991 V=800.0 PL=0
MOVL C00992 V=800.0 PL=0
MOVL C00993 V=800.0 PL=0
MOVL C00994 V=800.0 PL=0
MOVL C00995 V=800.0 PL=0
MOVL C00996 V=800.0 PL=0
MOVL C00997 V=800.0 PL=0
MOVL C00998 V=800.0 PL=0
MOVL C00999 V=800.0 PL=0
MOVL C01000 V=800.0 PL=0
MOVL C01001 V=800.0 PL=0
MOVL C01002 V=800.0 PL=0
MOVL C01003 V=800.0 PL=0
MOVL C01004 V=800.0 PL=0
MOVL C01005 V=800.0 PL=0
MOVL C01006 V=800.0 PL=0
MOVL C01007 V=800.0 PL=0
MOVL C01008 V=800.0 PL=0
MOVL C01009 V=800.0 PL=0
MOVL C01010 V=800.0 PL=0
MOVL C01011 V=800.0 PL=0
MOVL C01012 V=800.0 PL=0
MOVL C01013 V=800.0 PL=0
MOVL C01014 V=800.0 PL=0
MOVL C01015 V=800.0 PL=0
MOVL C01016 V=800.0 PL=0
MOVL C01017 V=800.0 PL=0
MOVL C01018 V=800.0 PL=0
MOVL C01019 V=800.0 PL=0
MOVL C01020 V=800.0 PL=0
MOVL C01021 V=800.0 PL=0
MOVL C01022 V=800.0 PL=0
MOVL C01023 V=800.0 PL=0
MOVL C01024 V=800.0 PL=0
MOVL C01025 V=800.0 PL=0
MOVL C01026 V=800.0 PL=0
MOVL C01027 V=800.0 PL=0
MOVL C01028 V=800.0 PL=0
MOVL C01029 V=800.0 PL=0
MOVL C01030 V=800.0 PL=0
MOVL C01031 V=800.0 PL=0
MOVL C01032 V=800.0 PL=0
MOVL C01033 V=800.0 PL=0
MOVL C01034 V=800.0 PL=0
MOVL C01035 V=800.0 PL=0
MOVL C01036 V=800.0 PL=0
MOVL C01037 V=800.0 PL=0
MOVL C01038 V=800.0 PL=0
MOVL C01039 V=800.0 PL=0
MOVL C01040 V=800.0 PL=0
MOVL C01041 V=800.0 PL=0
MOVL C01042 V=800.0 PL=0
MOVL C01043 V=800.0 PL=0
MOVL C01044 V=800.0 PL=0
MOVL C01045 V=800.0 PL=0
MOVL C01046 V=800.0 PL=0
MOVL C01047 V=800.0 PL=0
MOVL C01048 V=800.0 PL=0
MOVL C01049 V=800.0 PL=0
MOVL C01050 V=800.0 PL=0
MOVL C01051 V=800.0 PL=0
MOVL C01052 V=800.0 PL=0
MOVL C01053 V=800.0 PL=0
MOVL C01054 V=800.0 PL=0
MOVL C01055 V=800.0 PL=0
MOVL C01056 V=800.0 PL=0
MOVL C01057 V=800.0 PL=0
MOVL C01058 V=800.0 PL=0
MOVL C01059 V=800.0 PL=0
MOVL C01060 V=800.0 PL=0
MOVL C01061 V=800.0 PL=0
MOVL C01062 V=800.0 PL=0
MOVL C01063 V=800.0 PL=0
MOVL C01064 V=800.0 PL=0
MOVL C01065 V=800.0 PL=0
MOVL C01066 V=800.0 PL=0
MOVL C01067 V=800.0 PL=0
MOVL C01068 V=800.0 PL=0
MOVL C01069 V=800.0 PL=0
MOVL C01070 V=800.0 PL=0
MOVL C01071 V=800.0 PL=0
MOVL C01072 V=800.0 PL=0
MOVL C01073 V=800.0 PL=0
MOVL C01074 V=800.0 PL=0
MOVL C01075 V=800.0 PL=0
MOVL C01076 V=800.0 PL=0
MOVL C01077 V=800.0 PL=0
MOVL C01078 V=800.0 PL=0
MOVL C01079 V=800.0 PL=0
MOVL C01080 V=800.0 PL=0
MOVL C01081 V=800.0 PL=0
MOVL C01082 V=800.0 PL=0
MOVL C01083 V=800.0 PL=0
MOVL C01084 V=800.0 PL=0
MOVL C01085 V=800.0 PL=0
MOVL C01086 V=800.0 PL=0
MOVL C01087 V=800.0 PL=0
MOVL C01088 V=800.0 PL=0
MOVL C01089 V=800.0 PL=0
MOVL C01090 V=800.0 PL=0
MOVL C01091 V=800.0 PL=0
MOVL C01092 V=800.0 PL=0
MOVL C01093 V=800.0 PL=0
MOVL C01094 V=800.0 PL=0
MOVL C01095 V=800.0 PL=0
MOVL C01096 V=800.0 PL=0
MOVL C01097 V=800.0 PL=0
MOVL C01098 V=800.0 PL=0
MOVL C01099 V=800.0 PL=0
MOVL C01100 V=800.0 PL=0
MOVL C01101 V=800.0 PL=0
MOVL C01102 V=800.0 PL=0
MOVL C01103 V=800.0 PL=0
MOVL C01104 V=800.0 PL=0
MOVL C01105 V=800.0 PL=0
MOVL C01106 V=800.0 PL=0
MOVL C01107 V=800.0 PL=0
MOVL C01108 V=800.0 PL=0
MOVL C01109 V=800.0 PL=0
MOVL C01110 V=800.0 PL=0
MOVL C01111 V=800.0 PL=0
MOVL C01112 V=800.0 PL=0
MOVL C01113 V=800.0 PL=0
MOVL C01114 V=800.0 PL=0
MOVL C01115 V=800.0 PL=0
MOVL C01116 V=800.0 PL=0
MOVL C01117 V=800.0 PL=0
MOVL C01118 V=800.0 PL=0
MOVL C01119 V=800.0 PL=0
MOVL C01120 V=800.0 PL=0
MOVL C01121 V=800.0 PL=0
MOVL C01122 V=800.0 PL=0
MOVL C01123 V=800.0 PL=0
MOVL C01124 V=800.0 PL=0
MOVL C01125 V=800.0 PL=0
MOVL C01126 V=800.0 PL=0
MOVL C01127 V=800.0 PL=0
MOVL C01128 V=800.0 PL=0
MOVL C01129 V=800.0 PL=0
MOVL C01130 V=800.0 PL=0
MOVL C01131 V=800.0 PL=0
MOVL C01132 V=800.0 PL=0
MOVL C01133 V=800.0 PL=0
MOVL C01134 V=800.0 PL=0
MOVL C01135 V=800.0 PL=0
MOVL C01136 V=800.0 PL=0
MOVL C01137 V=800.0 PL=0
MOVL C01138 V=800.0 PL=0
MOVL C01139 V=800.0 PL=0
MOVL C01140 V=800.0 PL=0
MOVL C01141 V=800.0 PL=0
MOVL C01142 V=800.0 PL=0
MOVL C01143 V=800.0 PL=0
MOVL C01144 V=800.0 PL=0
MOVL C01145 V=800.0 PL=0
MOVL C01146 V=800.0 PL=0
MOVL C01147 V=800.0 PL=0
MOVL C01148 V=800.0 PL=0
MOVL C01149 V=800.0 PL=0
MOVL C01150 V=800.0 PL=0
MOVL C01151 V=800.0 PL=0
MOVL C01152 V=800.0 PL=0
MOVL C01153 V=800.0 PL=0
MOVL C01154 V=800.0 PL=0
MOVL C01155 V=800.0 PL=0
MOVL C01156 V=800.0 PL=0
MOVL C01157 V=800.0 PL=0
MOVL C01158 V=800.0 PL=0
MOVL C01159 V=800.0 PL=0
MOVL C01160 V=800.0 PL=0
MOVL C01161 V=800.0 PL=0
MOVL C01162 V=800.0 PL=0
MOVL C01163 V=800.0 PL=0
MOVL C01164 V=800.0 PL=0
MOVL C01165 V=800.0 PL=0
MOVL C01166 V=800.0 PL=0
MOVL C01167 V=800.0 PL=0
MOVL C01168 V=800.0 PL=0
MOVL C01169 V=800.0 PL=0
MOVL C01170 V=800.0 PL=0
MOVL C01171 V=800.0 PL=0
MOVL C01172 V=800.0 PL=0
MOVL C01173 V=800.0 PL=0
MOVL C01174 V=800.0 PL=0
MOVL C01175 V=800.0 PL=0
MOVL C01176 V=800.0 PL=0
MOVL C01177 V=800.0 PL=0
MOVL C01178 V=800.0 PL=0
MOVL C01179 V=800.0 PL=0
MOVL C01180 V=800.0 PL=0
MOVL C01181 V=800.0 PL=0
MOVL C01182 V=800.0 PL=0
MOVL C01183 V=800.0 PL=0
MOVL C01184 V=800.0 PL=0
MOVL C01185 V=800.0 PL=0
MOVL C01186 V=800.0 PL=0
MOVL C01187 V=800.0 PL=0
MOVL C01188 V=800.0 PL=0
MOVL C01189 V=800.0 PL=0
MOVL C01190 V=800.0 PL=0
MOVL C01191 V=800.0 PL=0
MOVL C01192 V=800.0 PL=0
MOVL C01193 V=800.0 PL=0
MOVL C01194 V=800.0 PL=0
MOVL C01195 V=800.0 PL=0
MOVL C01196 V=800.0 PL=0
MOVL C01197 V=800.0 PL=0
MOVL C01198 V=800.0 PL=0
MOVL C01199 V=800.0 PL=0
MOVL C01200 V=800.0 PL=0
MOVL C01201 V=800.0 PL=0
MOVL C01202 V=800.0 PL=0
MOVL C01203 V=800.0 PL=0
MOVL C01204 V=800.0 PL=0
MOVL C01205 V=800.0 PL=0
MOVL C01206 V=800.0 PL=0
MOVL C01207 V=800.0 PL=0
MOVL C01208 V=800.0 PL=0
MOVL C01209 V=800.0 PL=0
MOVL C01210 V=800.0 PL=0
MOVL C01211 V=800.0 PL=0
MOVL C01212 V=800.0 PL=0
MOVL C01213 V=800.0 PL=0
MOVL C01214 V=800.0 PL=0
MOVL C01215 V=800.0 PL=0
MOVL C01216 V=800.0 PL=0
MOVL C01217 V=800.0 PL=0
MOVL C01218 V=800.0 PL=0
MOVL C01219 V=800.0 PL=0
MOVL C01220 V=800.0 PL=0
MOVL C01221 V=800.0 PL=0
MOVL C01222 V=800.0 PL=0
MOVL C01223 V=800.0 PL=0
MOVL C01224 V=800.0 PL=0
MOVL C01225 V=800.0 PL=0
MOVL C01226 V=800.0 PL=0
MOVL C01227 V=800.0 PL=0
MOVL C01228 V=800.0 PL=0
MOVL C01229 V=800.0 PL=0
MOVL C01230 V=800.0 PL=0
MOVL C01231 V=800.0 PL=0
MOVL C01232 V=800.0 PL=0
MOVL C01233 V=800.0 PL=0
MOVL C01234 V=800.0 PL=0
MOVL C01235 V=800.0 PL=0
MOVL C01236 V=800.0 PL=0
MOVL C01237 V=800.0 PL=0
MOVL C01238 V=800.0 PL=0
MOVL C01239 V=800.0 PL=0
MOVL C01240 V=800.0 PL=0
MOVL C01241 V=800.0 PL=0
MOVL C01242 V=800.0 PL=0
MOVL C01243 V=800.0 PL=0
MOVL C01244 V=800.0 PL=0
MOVL C01245 V=800.0 PL=0
MOVL C01246 V=800.0 PL=0
MOVL C01247 V=800.0 PL=0
MOVL C01248 V=800.0 PL=0
MOVL C01249 V=800.0 PL=0
MOVL C01250 V=800.0 PL=0
MOVL C01251 V=800.0 PL=0
MOVL C01252 V=800.0 PL=0
MOVL C01253 V=800.0 PL=0
MOVL C01254 V=800.0 PL=0
MOVL C01255 V=800.0 PL=0
MOVL C01256 V=800.0 PL=0
MOVL C01257 V=800.0 PL=0
MOVL C01258 V=800.0 PL=0
MOVL C01259 V=800.0 PL=0
MOVL C01260 V=800.0 PL=0
MOVL C01261 V=800.0 PL=0
MOVL C01262 V=800.0 PL=0
MOVL C01263 V=800.0 PL=0
MOVL C01264 V=800.0 PL=0
MOVL C01265 V=800.0 PL=0
MOVL C01266 V=800.0 PL=0
MOVL C01267 V=800.0 PL=0
MOVL C01268 V=800.0 PL=0
MOVL C01269 V=800.0 PL=0
MOVL C01270 V=800.0 PL=0
MOVL C01271 V=800.0 PL=0
MOVL C01272 V=800.0 PL=0
MOVL C01273 V=800.0 PL=0
MOVL C01274 V=800.0 PL=0
MOVL C01275 V=800.0 PL=0
MOVL C01276 V=800.0 PL=0
MOVL C01277 V=800.0 PL=0
MOVL C01278 V=800.0 PL=0
MOVL C01279 V=800.0 PL=0
MOVL C01280 V=800.0 PL=0
MOVL C01281 V=800.0 PL=0
MOVL C01282 V=800.0 PL=0
MOVL C01283 V=800.0 PL=0
MOVL C01284 V=800.0 PL=0
MOVL C01285 V=800.0 PL=0
MOVL C01286 V=800.0 PL=0
MOVL C01287 V=800.0 PL=0
MOVL C01288 V=800.0 PL=0
MOVL C01289 V=800.0 PL=0
MOVL C01290 V=800.0 PL=0
MOVL C01291 V=800.0 PL=0
MOVL C01292 V=800.0 PL=0
MOVL C01293 V=800.0 PL=0
MOVL C01294 V=800.0 PL=0
MOVL C01295 V=800.0 PL=0
MOVL C01296 V=800.0 PL=0
MOVL C01297 V=800.0 PL=0
MOVL C01298 V=800.0 PL=0
MOVL C01299 V=800.0 PL=0
MOVL C01300 V=800.0 PL=0
MOVL C01301 V=800.0 PL=0
MOVL C01302 V=800.0 PL=0
MOVL C01303 V=800.0 PL=0
MOVL C01304 V=800.0 PL=0
MOVL C01305 V=800.0 PL=0
MOVL C01306 V=800.0 PL=0
MOVL C01307 V=800.0 PL=0
MOVL C01308 V=800.0 PL=0
MOVL C01309 V=800.0 PL=0
MOVL C01310 V=800.0 PL=0
MOVL C01311 V=800.0 PL=0
MOVL C01312 V=800.0 PL=0
MOVL C01313 V=800.0 PL=0
MOVL C01314 V=800.0 PL=0
MOVL C01315 V=800.0 PL=0
MOVL C01316 V=800.0 PL=0
MOVL C01317 V=800.0 PL=0
MOVL C01318 V=800.0 PL=0
MOVL C01319 V=800.0 PL=0
MOVL C01320 V=800.0 PL=0
MOVL C01321 V=800.0 PL=0
MOVL C01322 V=800.0 PL=0
MOVL C01323 V=800.0 PL=0
MOVL C01324 V=800.0 PL=0
MOVL C01325 V=800.0 PL=0
MOVL C01326 V=800.0 PL=0
MOVL C01327 V=800.0 PL=0
MOVL C01328 V=800.0 PL=0
MOVL C01329 V=800.0 PL=0
MOVL C01330 V=800.0 PL=0
MOVL C01331 V=800.0 PL=0
MOVL C01332 V=800.0 PL=0
MOVL C01333 V=800.0 PL=0
MOVL C01334 V=800.0 PL=0
MOVL C01335 V=800.0 PL=0
MOVL C01336 V=800.0 PL=0
MOVL C01337 V=800.0 PL=0
MOVL C01338 V=800.0 PL=0
MOVL C01339 V=800.0 PL=0
MOVL C01340 V=800.0 PL=0
MOVL C01341 V=800.0 PL=0
MOVL C01342 V=800.0 PL=0
MOVL C01343 V=800.0 PL=0
MOVL C01344 V=800.0 PL=0
MOVL C01345 V=800.0 PL=0
MOVL C01346 V=800.0 PL=0
MOVL C01347 V=800.0 PL=0
MOVL C01348 V=800.0 PL=0
MOVL C01349 V=800.0 PL=0
MOVL C01350 V=800.0 PL=0
MOVL C01351 V=800.0 PL=0
MOVL C01352 V=800.0 PL=0
MOVL C01353 V=800.0 PL=0
MOVL C01354 V=800.0 PL=0
MOVL C01355 V=800.0 PL=0
MOVL C01356 V=800.0 PL=0
MOVL C01357 V=800.0 PL=0
MOVL C01358 V=800.0 PL=0
MOVL C01359 V=800.0 PL=0
MOVL C01360 V=800.0 PL=0
MOVL C01361 V=800.0 PL=0
MOVL C01362 V=800.0 PL=0
MOVL C01363 V=800.0 PL=0
MOVL C01364 V=800.0 PL=0
MOVL C01365 V=800.0 PL=0
MOVL C01366 V=800.0 PL=0
MOVL C01367 V=800.0 PL=0
MOVL C01368 V=800.0 PL=0
MOVL C01369 V=800.0 PL=0
MOVL C01370 V=800.0 PL=0
MOVL C01371 V=800.0 PL=0
MOVL C01372 V=800.0 PL=0
MOVL C01373 V=800.0 PL=0
MOVL C01374 V=800.0 PL=0
MOVL C01375 V=800.0 PL=0
MOVL C01376 V=800.0 PL=0
MOVL C01377 V=800.0 PL=0
MOVL C01378 V=800.0 PL=0
MOVL C01379 V=800.0 PL=0
MOVL C01380 V=800.0 PL=0
MOVL C01381 V=800.0 PL=0
MOVL C01382 V=800.0 PL=0
MOVL C01383 V=800.0 PL=0
MOVL C01384 V=800.0 PL=0
MOVL C01385 V=800.0 PL=0
MOVL C01386 V=800.0 PL=0
MOVL C01387 V=800.0 PL=0
MOVL C01388 V=800.0 PL=0
MOVL C01389 V=800.0 PL=0
MOVL C01390 V=800.0 PL=0
MOVL C01391 V=800.0 PL=0
MOVL C01392 V=800.0 PL=0
MOVL C01393 V=800.0 PL=0
MOVL C01394 V=800.0 PL=0
MOVL C01395 V=800.0 PL=0
MOVL C01396 V=800.0 PL=0
MOVL C01397 V=800.0 PL=0
MOVL C01398 V=800.0 PL=0
MOVL C01399 V=800.0 PL=0
MOVL C01400 V=800.0 PL=0
MOVL C01401 V=800.0 PL=0
MOVL C01402 V=800.0 PL=0
MOVL C01403 V=800.0 PL=0
MOVL C01404 V=800.0 PL=0
MOVL C01405 V=800.0 PL=0
MOVL C01406 V=800.0 PL=0
MOVL C01407 V=800.0 PL=0
MOVL C01408 V=800.0 PL=0
MOVL C01409 V=800.0 PL=0
MOVL C01410 V=800.0 PL=0
MOVL C01411 V=800.0 PL=0
MOVL C01412 V=800.0 PL=0
MOVL C01413 V=800.0 PL=0
MOVL C01414 V=800.0 PL=0
MOVL C01415 V=800.0 PL=0
MOVL C01416 V=800.0 PL=0
MOVL C01417 V=800.0 PL=0
MOVL C01418 V=800.0 PL=0
MOVL C01419 V=800.0 PL=0
MOVL C01420 V=800.0 PL=0
MOVL C01421 V=800.0 PL=0
MOVL C01422 V=800.0 PL=0
MOVL C01423 V=800.0 PL=0
MOVL C01424 V=800.0 PL=0
MOVL C01425 V=800.0 PL=0
MOVL C01426 V=800.0 PL=0
MOVL C01427 V=800.0 PL=0
MOVL C01428 V=800.0 PL=0
MOVL C01429 V=800.0 PL=0
MOVL C01430 V=800.0 PL=0
MOVL C01431 V=800.0 PL=0
MOVL C01432 V=800.0 PL=0
MOVL C01433 V=800.0 PL=0
MOVL C01434 V=800.0 PL=0
MOVL C01435 V=800.0 PL=0
MOVL C01436 V=800.0 PL=0
MOVL C01437 V=800.0 PL=0
MOVL C01438 V=800.0 PL=0
MOVL C01439 V=800.0 PL=0
MOVL C01440 V=800.0 PL=0
MOVL C01441 V=800.0 PL=0
MOVL C01442 V=800.0 PL=0
MOVL C01443 V=800.0 PL=0
MOVL C01444 V=800.0 PL=0
MOVL C01445 V=800.0 PL=0
MOVL C01446 V=800.0 PL=0
MOVL C01447 V=800.0 PL=0
MOVL C01448 V=800.0 PL=0
MOVL C01449 V=800.0 PL=0
MOVL C01450 V=800.0 PL=0
MOVL C01451 V=800.0 PL=0
MOVL C01452 V=800.0 PL=0
MOVL C01453 V=800.0 PL=0
MOVL C01454 V=800.0 PL=0
MOVL C01455 V=800.0 PL=0
MOVL C01456 V=800.0 PL=0
MOVL C01457 V=800.0 PL=0
MOVL C01458 V=800.0 PL=0
MOVL C01459 V=800.0 PL=0
MOVL C01460 V=800.0 PL=0
MOVL C01461 V=800.0 PL=0
MOVL C01462 V=800.0 PL=0
MOVL C01463 V=800.0 PL=0
MOVL C01464 V=800.0 PL=0
MOVL C01465 V=800.0 PL=0
MOVL C01466 V=800.0 PL=0
MOVL C01467 V=800.0 PL=0
MOVL C01468 V=800.0 PL=0
MOVL C01469 V=800.0 PL=0
MOVL C01470 V=800.0 PL=0
MOVL C01471 V=800.0 PL=0
MOVL C01472 V=800.0 PL=0
MOVL C01473 V=800.0 PL=0
MOVL C01474 V=800.0 PL=0
MOVL C01475 V=800.0 PL=0
MOVL C01476 V=800.0 PL=0
MOVL C01477 V=800.0 PL=0
MOVL C01478 V=800.0 PL=0
MOVL C01479 V=800.0 PL=0
MOVL C01480 V=800.0 PL=0
MOVL C01481 V=800.0 PL=0
MOVL C01482 V=800.0 PL=0
MOVL C01483 V=800.0 PL=0
MOVL C01484 V=800.0 PL=0
MOVL C01485 V=800.0 PL=0
MOVL C01486 V=800.0 PL=0
MOVL C01487 V=800.0 PL=0
MOVL C01488 V=800.0 PL=0
MOVL C01489 V=800.0 PL=0
MOVL C01490 V=800.0 PL=0
MOVL C01491 V=800.0 PL=0
MOVL C01492 V=800.0 PL=0
MOVL C01493 V=800.0 PL=0
MOVL C01494 V=800.0 PL=0
MOVL C01495 V=800.0 PL=0
MOVL C01496 V=800.0 PL=0
MOVL C01497 V=800.0 PL=0
MOVL C01498 V=800.0 PL=0
MOVL C01499 V=800.0 PL=0
MOVL C01500 V=800.0 PL=0
MOVL C01501 V=800.0 PL=0
MOVL C01502 V=800.0 PL=0
MOVL C01503 V=800.0 PL=0
MOVL C01504 V=800.0 PL=0
MOVL C01505 V=800.0 PL=0
MOVL C01506 V=800.0 PL=0
MOVL C01507 V=800.0 PL=0
MOVL C01508 V=800.0 PL=0
MOVL C01509 V=800.0 PL=0
MOVL C01510 V=800.0 PL=0
MOVL C01511 V=800.0 PL=0
MOVL C01512 V=800.0 PL=0
MOVL C01513 V=800.0 PL=0
MOVL C01514 V=800.0 PL=0
MOVL C01515 V=800.0 PL=0
MOVL C01516 V=800.0 PL=0
MOVL C01517 V=800.0 PL=0
MOVL C01518 V=800.0 PL=0
MOVL C01519 V=800.0 PL=0
MOVL C01520 V=800.0 PL=0
MOVL C01521 V=800.0 PL=0
MOVL C01522 V=800.0 PL=0
MOVL C01523 V=800.0 PL=0
MOVL C01524 V=800.0 PL=0
MOVL C01525 V=800.0 PL=0
MOVL C01526 V=800.0 PL=0
MOVL C01527 V=800.0 PL=0
MOVL C01528 V=800.0 PL=0
MOVL C01529 V=800.0 PL=0
MOVL C01530 V=800.0 PL=0
MOVL C01531 V=800.0 PL=0
MOVL C01532 V=800.0 PL=0
MOVL C01533 V=800.0 PL=0
MOVL C01534 V=800.0 PL=0
MOVL C01535 V=800.0 PL=0
MOVL C01536 V=800.0 PL=0
MOVL C01537 V=800.0 PL=0
MOVL C01538 V=800.0 PL=0
MOVL C01539 V=800.0 PL=0
MOVL C01540 V=800.0 PL=0
MOVL C01541 V=800.0 PL=0
MOVL C01542 V=800.0 PL=0
MOVL C01543 V=800.0 PL=0
MOVL C01544 V=800.0 PL=0
MOVL C01545 V=800.0 PL=0
MOVL C01546 V=800.0 PL=0
MOVL C01547 V=800.0 PL=0
MOVL C01548 V=800.0 PL=0
MOVL C01549 V=800.0 PL=0
MOVL C01550 V=800.0 PL=0
MOVL C01551 V=800.0 PL=0
MOVL C01552 V=800.0 PL=0
MOVL C01553 V=800.0 PL=0
MOVL C01554 V=800.0 PL=0
MOVL C01555 V=800.0 PL=0
MOVL C01556 V=800.0 PL=0
MOVL C01557 V=800.0 PL=0
MOVL C01558 V=800.0 PL=0
MOVL C01559 V=800.0 PL=0
MOVL C01560 V=800.0 PL=0
MOVL C01561 V=800.0 PL=0
MOVL C01562 V=800.0 PL=0
MOVL C01563 V=800.0 PL=0
MOVL C01564 V=800.0 PL=0
MOVL C01565 V=800.0 PL=0
MOVL C01566 V=800.0 PL=0
MOVL C01567 V=800.0 PL=0
MOVL C01568 V=800.0 PL=0
MOVL C01569 V=800.0 PL=0
MOVL C01570 V=800.0 PL=0
MOVL C01571 V=800.0 PL=0
MOVL C01572 V=800.0 PL=0
MOVL C01573 V=800.0 PL=0
MOVL C01574 V=800.0 PL=0
MOVL C01575 V=800.0 PL=0
MOVL C01576 V=800.0 PL=0
MOVL C01577 V=800.0 PL=0
MOVL C01578 V=800.0 PL=0
MOVL C01579 V=800.0 PL=0
MOVL C01580 V=800.0 PL=0
MOVL C01581 V=800.0 PL=0
MOVL C01582 V=800.0 PL=0
MOVL C01583 V=800.0 PL=0
MOVL C01584 V=800.0 PL=0
MOVL C01585 V=800.0 PL=0
MOVL C01586 V=800.0 PL=0
MOVL C01587 V=800.0 PL=0
MOVL C01588 V=800.0 PL=0
MOVL C01589 V=800.0 PL=0
MOVL C01590 V=800.0 PL=0
MOVL C01591 V=800.0 PL=0
MOVL C01592 V=800.0 PL=0
MOVL C01593 V=800.0 PL=0
MOVL C01594 V=800.0 PL=0
MOVL C01595 V=800.0 PL=0
MOVL C01596 V=800.0 PL=0
MOVL C01597 V=800.0 PL=0
MOVL C01598 V=800.0 PL=0
MOVL C01599 V=800.0 PL=0
MOVL C01600 V=800.0 PL=0
MOVL C01601 V=800.0 PL=0
MOVL C01602 V=800.0 PL=0
MOVL C01603 V=800.0 PL=0
MOVL C01604 V=800.0 PL=0
MOVL C01605 V=800.0 PL=0
MOVL C01606 V=800.0 PL=0
MOVL C01607 V=800.0 PL=0
MOVL C01608 V=800.0 PL=0
MOVL C01609 V=800.0 PL=0
MOVL C01610 V=800.0 PL=0
MOVL C01611 V=800.0 PL=0
MOVL C01612 V=800.0 PL=0
MOVL C01613 V=800.0 PL=0
MOVL C01614 V=800.0 PL=0
MOVL C01615 V=800.0 PL=0
MOVL C01616 V=800.0 PL=0
MOVL C01617 V=800.0 PL=0
MOVL C01618 V=800.0 PL=0
MOVL C01619 V=800.0 PL=0
MOVL C01620 V=800.0 PL=0
MOVL C01621 V=800.0 PL=0
MOVL C01622 V=800.0 PL=0
MOVL C01623 V=800.0 PL=0
MOVL C01624 V=800.0 PL=0
MOVL C01625 V=800.0 PL=0
MOVL C01626 V=800.0 PL=0
MOVL C01627 V=800.0 PL=0
MOVL C01628 V=800.0 PL=0
MOVL C01629 V=800.0 PL=0
MOVL C01630 V=800.0 PL=0
MOVL C01631 V=800.0 PL=0
MOVL C01632 V=800.0 PL=0
MOVL C01633 V=800.0 PL=0
MOVL C01634 V=800.0 PL=0
MOVL C01635 V=800.0 PL=0
MOVL C01636 V=800.0 PL=0
MOVL C01637 V=800.0 PL=0
MOVL C01638 V=800.0 PL=0
MOVL C01639 V=800.0 PL=0
MOVL C01640 V=800.0 PL=0
MOVL C01641 V=800.0 PL=0
MOVL C01642 V=800.0 PL=0
MOVL C01643 V=800.0 PL=0
MOVL C01644 V=800.0 PL=0
MOVL C01645 V=800.0 PL=0
MOVL C01646 V=800.0 PL=0
MOVL C01647 V=800.0 PL=0
MOVL C01648 V=800.0 PL=0
MOVL C01649 V=800.0 PL=0
MOVL C01650 V=800.0 PL=0
MOVL C01651 V=800.0 PL=0
MOVL C01652 V=800.0 PL=0
MOVL C01653 V=800.0 PL=0
MOVL C01654 V=800.0 PL=0
MOVL C01655 V=800.0 PL=0
MOVL C01656 V=800.0 PL=0
MOVL C01657 V=800.0 PL=0
MOVL C01658 V=800.0 PL=0
MOVL C01659 V=800.0 PL=0
MOVL C01660 V=800.0 PL=0
MOVL C01661 V=800.0 PL=0
MOVL C01662 V=800.0 PL=0
MOVL C01663 V=800.0 PL=0
MOVL C01664 V=800.0 PL=0
MOVL C01665 V=800.0 PL=0
MOVL C01666 V=800.0 PL=0
MOVL C01667 V=800.0 PL=0
MOVL C01668 V=800.0 PL=0
MOVL C01669 V=800.0 PL=0
MOVL C01670 V=800.0 PL=0
MOVL C01671 V=800.0 PL=0
MOVL C01672 V=800.0 PL=0
MOVL C01673 V=800.0 PL=0
MOVL C01674 V=800.0 PL=0
MOVL C01675 V=800.0 PL=0
MOVL C01676 V=800.0 PL=0
MOVL C01677 V=800.0 PL=0
MOVL C01678 V=800.0 PL=0
MOVL C01679 V=800.0 PL=0
MOVL C01680 V=800.0 PL=0
MOVL C01681 V=800.0 PL=0
MOVL C01682 V=800.0 PL=0
MOVL C01683 V=800.0 PL=0
MOVL C01684 V=800.0 PL=0
MOVL C01685 V=800.0 PL=0
MOVL C01686 V=800.0 PL=0
MOVL C01687 V=800.0 PL=0
MOVL C01688 V=800.0 PL=0
MOVL C01689 V=800.0 PL=0
MOVL C01690 V=800.0 PL=0
MOVL C01691 V=800.0 PL=0
MOVL C01692 V=800.0 PL=0
MOVL C01693 V=800.0 PL=0
MOVL C01694 V=800.0 PL=0
MOVL C01695 V=800.0 PL=0
MOVL C01696 V=800.0 PL=0
MOVL C01697 V=800.0 PL=0
MOVL C01698 V=800.0 PL=0
MOVL C01699 V=800.0 PL=0
MOVL C01700 V=800.0 PL=0
MOVL C01701 V=800.0 PL=0
MOVL C01702 V=800.0 PL=0
MOVL C01703 V=800.0 PL=0
MOVL C01704 V=800.0 PL=0
MOVL C01705 V=800.0 PL=0
MOVL C01706 V=800.0 PL=0
MOVL C01707 V=800.0 PL=0
MOVL C01708 V=800.0 PL=0
MOVL C01709 V=800.0 PL=0
MOVL C01710 V=800.0 PL=0
MOVL C01711 V=800.0 PL=0
MOVL C01712 V=800.0 PL=0
MOVL C01713 V=800.0 PL=0
MOVL C01714 V=800.0 PL=0
MOVL C01715 V=800.0 PL=0
MOVL C01716 V=800.0 PL=0
MOVL C01717 V=800.0 PL=0
MOVL C01718 V=800.0 PL=0
MOVL C01719 V=800.0 PL=0
MOVL C01720 V=800.0 PL=0
MOVL C01721 V=800.0 PL=0
MOVL C01722 V=800.0 PL=0
MOVL C01723 V=800.0 PL=0
MOVL C01724 V=800.0 PL=0
MOVL C01725 V=800.0 PL=0
MOVL C01726 V=800.0 PL=0
MOVL C01727 V=800.0 PL=0
MOVL C01728 V=800.0 PL=0
MOVL C01729 V=800.0 PL=0
MOVL C01730 V=800.0 PL=0
MOVL C01731 V=800.0 PL=0
MOVL C01732 V=800.0 PL=0
MOVL C01733 V=800.0 PL=0
MOVL C01734 V=800.0 PL=0
MOVL C01735 V=800.0 PL=0
MOVL C01736 V=800.0 PL=0
MOVL C01737 V=800.0 PL=0
MOVL C01738 V=800.0 PL=0
MOVL C01739 V=800.0 PL=0
MOVL C01740 V=800.0 PL=0
MOVL C01741 V=800.0 PL=0
MOVL C01742 V=800.0 PL=0
MOVL C01743 V=800.0 PL=0
MOVL C01744 V=800.0 PL=0
MOVL C01745 V=800.0 PL=0
MOVL C01746 V=800.0 PL=0
MOVL C01747 V=800.0 PL=0
MOVL C01748 V=800.0 PL=0
MOVL C01749 V=800.0 PL=0
MOVL C01750 V=800.0 PL=0
MOVL C01751 V=800.0 PL=0
MOVL C01752 V=800.0 PL=0
MOVL C01753 V=800.0 PL=0
MOVL C01754 V=800.0 PL=0
MOVL C01755 V=800.0 PL=0
MOVL C01756 V=800.0 PL=0
MOVL C01757 V=800.0 PL=0
MOVL C01758 V=800.0 PL=0
MOVL C01759 V=800.0 PL=0
MOVL C01760 V=800.0 PL=0
MOVL C01761 V=800.0 PL=0
MOVL C01762 V=800.0 PL=0
MOVL C01763 V=800.0 PL=0
MOVL C01764 V=800.0 PL=0
MOVL C01765 V=800.0 PL=0
MOVL C01766 V=800.0 PL=0
MOVL C01767 V=800.0 PL=0
MOVL C01768 V=800.0 PL=0
MOVL C01769 V=800.0 PL=0
MOVL C01770 V=800.0 PL=0
MOVL C01771 V=800.0 PL=0
MOVL C01772 V=800.0 PL=0
MOVL C01773 V=800.0 PL=0
MOVL C01774 V=800.0 PL=0
MOVL C01775 V=800.0 PL=0
MOVL C01776 V=800.0 PL=0
MOVL C01777 V=800.0 PL=0
MOVL C01778 V=800.0 PL=0
MOVL C01779 V=800.0 PL=0
MOVL C01780 V=800.0 PL=0
MOVL C01781 V=800.0 PL=0
MOVL C01782 V=800.0 PL=0
MOVL C01783 V=800.0 PL=0
MOVL C01784 V=800.0 PL=0
MOVL C01785 V=800.0 PL=0
MOVL C01786 V=800.0 PL=0
MOVL C01787 V=800.0 PL=0
MOVL C01788 V=800.0 PL=0
MOVL C01789 V=800.0 PL=0
MOVL C01790 V=800.0 PL=0
MOVL C01791 V=800.0 PL=0
MOVL C01792 V=800.0 PL=0
MOVL C01793 V=800.0 PL=0
MOVL C01794 V=800.0 PL=0
MOVL C01795 V=800.0 PL=0
MOVL C01796 V=800.0 PL=0
MOVL C01797 V=800.0 PL=0
MOVL C01798 V=800.0 PL=0
MOVL C01799 V=800.0 PL=0
MOVL C01800 V=800.0 PL=0
MOVL C01801 V=800.0 PL=0
MOVL C01802 V=800.0 PL=0
MOVL C01803 V=800.0 PL=0
MOVL C01804 V=800.0 PL=0
MOVL C01805 V=800.0 PL=0
MOVL C01806 V=800.0 PL=0
MOVL C01807 V=800.0 PL=0
MOVL C01808 V=800.0 PL=0
MOVL C01809 V=800.0 PL=0
MOVL C01810 V=800.0 PL=0
MOVL C01811 V=800.0 PL=0
MOVL C01812 V=800.0 PL=0
MOVL C01813 V=800.0 PL=0
MOVL C01814 V=800.0 PL=0
MOVL C01815 V=800.0 PL=0
MOVL C01816 V=800.0 PL=0
MOVL C01817 V=800.0 PL=0
MOVL C01818 V=800.0 PL=0
MOVL C01819 V=800.0 PL=0
MOVL C01820 V=800.0 PL=0
MOVL C01821 V=800.0 PL=0
MOVL C01822 V=800.0 PL=0
MOVL C01823 V=800.0 PL=0
MOVL C01824 V=800.0 PL=0
MOVL C01825 V=800.0 PL=0
MOVL C01826 V=800.0 PL=0
MOVL C01827 V=800.0 PL=0
MOVL C01828 V=800.0 PL=0
MOVL C01829 V=800.0 PL=0
MOVL C01830 V=800.0 PL=0
MOVL C01831 V=800.0 PL=0
MOVL C01832 V=800.0 PL=0
MOVL C01833 V=800.0 PL=0
MOVL C01834 V=800.0 PL=0
MOVL C01835 V=800.0 PL=0
MOVL C01836 V=800.0 PL=0
MOVL C01837 V=800.0 PL=0
MOVL C01838 V=800.0 PL=0
MOVL C01839 V=800.0 PL=0
MOVL C01840 V=800.0 PL=0
MOVL C01841 V=800.0 PL=0
MOVL C01842 V=800.0 PL=0
MOVL C01843 V=800.0 PL=0
MOVL C01844 V=800.0 PL=0
MOVL C01845 V=800.0 PL=0
MOVL C01846 V=800.0 PL=0
MOVL C01847 V=800.0 PL=0
MOVL C01848 V=800.0 PL=0
MOVL C01849 V=800.0 PL=0
MOVL C01850 V=800.0 PL=0
MOVL C01851 V=800.0 PL=0
MOVL C01852 V=800.0 PL=0
MOVL C01853 V=800.0 PL=0
MOVL C01854 V=800.0 PL=0
MOVL C01855 V=800.0 PL=0
MOVL C01856 V=800.0 PL=0
MOVL C01857 V=800.0 PL=0
MOVL C01858 V=800.0 PL=0
MOVL C01859 V=800.0 PL=0
MOVL C01860 V=800.0 PL=0
MOVL C01861 V=800.0 PL=0
MOVL C01862 V=800.0 PL=0
MOVL C01863 V=800.0 PL=0
MOVL C01864 V=800.0 PL=0
MOVL C01865 V=800.0 PL=0
MOVL C01866 V=800.0 PL=0
MOVL C01867 V=800.0 PL=0
MOVL C01868 V=800.0 PL=0
MOVL C01869 V=800.0 PL=0
MOVL C01870 V=800.0 PL=0
MOVL C01871 V=800.0 PL=0
MOVL C01872 V=800.0 PL=0
MOVL C01873 V=800.0 PL=0
MOVL C01874 V=800.0 PL=0
MOVL C01875 V=800.0 PL=0
MOVL C01876 V=800.0 PL=0
MOVL C01877 V=800.0 PL=0
MOVL C01878 V=800.0 PL=0
MOVL C01879 V=800.0 PL=0
MOVL C01880 V=800.0 PL=0
MOVL C01881 V=800.0 PL=0
MOVL C01882 V=800.0 PL=0
MOVL C01883 V=800.0 PL=0
MOVL C01884 V=800.0 PL=0
MOVL C01885 V=800.0 PL=0
MOVL C01886 V=800.0 PL=0
MOVL C01887 V=800.0 PL=0
MOVL C01888 V=800.0 PL=0
MOVL C01889 V=800.0 PL=0
MOVL C01890 V=800.0 PL=0
MOVL C01891 V=800.0 PL=0
MOVL C01892 V=800.0 PL=0
MOVL C01893 V=800.0 PL=0
MOVL C01894 V=800.0 PL=0
MOVL C01895 V=800.0 PL=0
MOVL C01896 V=800.0 PL=0
MOVL C01897 V=800.0 PL=0
MOVL C01898 V=800.0 PL=0
MOVL C01899 V=800.0 PL=0
MOVL C01900 V=800.0 PL=0
MOVL C01901 V=800.0 PL=0
MOVL C01902 V=800.0 PL=0
MOVL C01903 V=800.0 PL=0
MOVL C01904 V=800.0 PL=0
MOVL C01905 V=800.0 PL=0
MOVL C01906 V=800.0 PL=0
MOVL C01907 V=800.0 PL=0
MOVL C01908 V=800.0 PL=0
MOVL C01909 V=800.0 PL=0
MOVL C01910 V=800.0 PL=0
MOVL C01911 V=800.0 PL=0
MOVL C01912 V=800.0 PL=0
MOVL C01913 V=800.0 PL=0
MOVL C01914 V=800.0 PL=0
MOVL C01915 V=800.0 PL=0
MOVL C01916 V=800.0 PL=0
MOVL C01917 V=800.0 PL=0
MOVL C01918 V=800.0 PL=0
MOVL C01919 V=800.0 PL=0
MOVL C01920 V=800.0 PL=0
MOVL C01921 V=800.0 PL=0
MOVL C01922 V=800.0 PL=0
MOVL C01923 V=800.0 PL=0
MOVL C01924 V=800.0 PL=0
MOVL C01925 V=800.0 PL=0
MOVL C01926 V=800.0 PL=0
MOVL C01927 V=800.0 PL=0
MOVL C01928 V=800.0 PL=0
MOVL C01929 V=800.0 PL=0
MOVL C01930 V=800.0 PL=0
MOVL C01931 V=800.0 PL=0
MOVL C01932 V=800.0 PL=0
MOVL C01933 V=800.0 PL=0
MOVL C01934 V=800.0 PL=0
MOVL C01935 V=800.0 PL=0
MOVL C01936 V=800.0 PL=0
MOVL C01937 V=800.0 PL=0
MOVL C01938 V=800.0 PL=0
MOVL C01939 V=800.0 PL=0
MOVL C01940 V=800.0 PL=0
MOVL C01941 V=800.0 PL=0
MOVL C01942 V=800.0 PL=0
MOVL C01943 V=800.0 PL=0
MOVL C01944 V=800.0 PL=0
MOVL C01945 V=800.0 PL=0
MOVL C01946 V=800.0 PL=0
MOVL C01947 V=800.0 PL=0
MOVL C01948 V=800.0 PL=0
MOVL C01949 V=800.0 PL=0
MOVL C01950 V=800.0 PL=0
MOVL C01951 V=800.0 PL=0
MOVL C01952 V=800.0 PL=0
MOVL C01953 V=800.0 PL=0
MOVL C01954 V=800.0 PL=0
MOVL C01955 V=800.0 PL=0
MOVL C01956 V=800.0 PL=0
MOVL C01957 V=800.0 PL=0
MOVL C01958 V=800.0 PL=0
MOVL C01959 V=800.0 PL=0
MOVL C01960 V=800.0 PL=0
MOVL C01961 V=800.0 PL=0
MOVL C01962 V=800.0 PL=0
MOVL C01963 V=800.0 PL=0
MOVL C01964 V=800.0 PL=0
MOVL C01965 V=800.0 PL=0
MOVL C01966 V=800.0 PL=0
MOVL C01967 V=800.0 PL=0
MOVL C01968 V=800.0 PL=0
MOVL C01969 V=800.0 PL=0
MOVL C01970 V=800.0 PL=0
MOVL C01971 V=800.0 PL=0
MOVL C01972 V=800.0 PL=0
MOVL C01973 V=800.0 PL=0
MOVL C01974 V=800.0 PL=0
MOVL C01975 V=800.0 PL=0
MOVL C01976 V=800.0 PL=0
MOVL C01977 V=800.0 PL=0
MOVL C01978 V=800.0 PL=0
MOVL C01979 V=800.0 PL=0
MOVL C01980 V=800.0 PL=0
MOVL C01981 V=800.0 PL=0
MOVL C01982 V=800.0 PL=0
MOVL C01983 V=800.0 PL=0
MOVL C01984 V=800.0 PL=0
MOVL C01985 V=800.0 PL=0
MOVL C01986 V=800.0 PL=0
MOVL C01987 V=800.0 PL=0
MOVL C01988 V=800.0 PL=0
MOVL C01989 V=800.0 PL=0
MOVL C01990 V=800.0 PL=0
MOVL C01991 V=800.0 PL=0
MOVL C01992 V=800.0 PL=0
MOVL C01993 V=800.0 PL=0
MOVL C01994 V=800.0 PL=0
MOVL C01995 V=800.0 PL=0
MOVL C01996 V=800.0 PL=0
MOVL C01997 V=800.0 PL=0
MOVL C01998 V=800.0 PL=0
MOVL C01999 V=800.0 PL=0
MOVL C02000 V=800.0 PL=0
MOVL C02001 V=800.0 PL=0
MOVL C02002 V=800.0 PL=0
MOVL C02003 V=800.0 PL=0
MOVL C02004 V=800.0 PL=0
MOVL C02005 V=800.0 PL=0
MOVL C02006 V=800.0 PL=0
MOVL C02007 V=800.0 PL=0
MOVL C02008 V=800.0 PL=0
MOVL C02009 V=800.0 PL=0
MOVL C02010 V=800.0 PL=0
MOVL C02011 V=800.0 PL=0
MOVL C02012 V=800.0 PL=0
MOVL C02013 V=800.0 PL=0
MOVL C02014 V=800.0 PL=0
MOVL C02015 V=800.0 PL=0
MOVL C02016 V=800.0 PL=0
MOVL C02017 V=800.0 PL=0
MOVL C02018 V=800.0 PL=0
MOVL C02019 V=800.0 PL=0
MOVL C02020 V=800.0 PL=0
MOVL C02021 V=800.0 PL=0
MOVL C02022 V=800.0 PL=0
MOVL C02023 V=800.0 PL=0
MOVL C02024 V=800.0 PL=0
MOVL C02025 V=800.0 PL=0
MOVL C02026 V=800.0 PL=0
MOVL C02027 V=800.0 PL=0
MOVL C02028 V=800.0 PL=0
MOVL C02029 V=800.0 PL=0
MOVL C02030 V=800.0 PL=0
MOVL C02031 V=800.0 PL=0
MOVL C02032 V=800.0 PL=0
MOVL C02033 V=800.0 PL=0
MOVL C02034 V=800.0 PL=0
MOVL C02035 V=800.0 PL=0
MOVL C02036 V=800.0 PL=0
MOVL C02037 V=800.0 PL=0
MOVL C02038 V=800.0 PL=0
MOVL C02039 V=800.0 PL=0
MOVL C02040 V=800.0 PL=0
MOVL C02041 V=800.0 PL=0
MOVL C02042 V=800.0 PL=0
MOVL C02043 V=800.0 PL=0
MOVL C02044 V=800.0 PL=0
MOVL C02045 V=800.0 PL=0
MOVL C02046 V=800.0 PL=0
MOVL C02047 V=800.0 PL=0
MOVL C02048 V=800.0 PL=0
MOVL C02049 V=800.0 PL=0
MOVL C02050 V=800.0 PL=0
MOVL C02051 V=800.0 PL=0
MOVL C02052 V=800.0 PL=0
MOVL C02053 V=800.0 PL=0
MOVL C02054 V=800.0 PL=0
MOVL C02055 V=800.0 PL=0
MOVL C02056 V=800.0 PL=0
MOVL C02057 V=800.0 PL=0
MOVL C02058 V=800.0 PL=0
MOVL C02059 V=800.0 PL=0
MOVL C02060 V=800.0 PL=0
MOVL C02061 V=800.0 PL=0
MOVL C02062 V=800.0 PL=0
MOVL C02063 V=800.0 PL=0
MOVL C02064 V=800.0 PL=0
MOVL C02065 V=800.0 PL=0
MOVL C02066 V=800.0 PL=0
MOVL C02067 V=800.0 PL=0
MOVL C02068 V=800.0 PL=0
MOVL C02069 V=800.0 PL=0
MOVL C02070 V=800.0 PL=0
MOVL C02071 V=800.0 PL=0
MOVL C02072 V=800.0 PL=0
MOVL C02073 V=800.0 PL=0
MOVL C02074 V=800.0 PL=0
MOVL C02075 V=800.0 PL=0
MOVL C02076 V=800.0 PL=0
MOVL C02077 V=800.0 PL=0
MOVL C02078 V=800.0 PL=0
MOVL C02079 V=800.0 PL=0
MOVL C02080 V=800.0 PL=0
MOVL C02081 V=800.0 PL=0
MOVL C02082 V=800.0 PL=0
MOVL C02083 V=800.0 PL=0
MOVL C02084 V=800.0 PL=0
MOVL C02085 V=800.0 PL=0
MOVL C02086 V=800.0 PL=0
MOVL C02087 V=800.0 PL=0
MOVL C02088 V=800.0 PL=0
MOVL C02089 V=800.0 PL=0
MOVL C02090 V=800.0 PL=0
MOVL C02091 V=800.0 PL=0
MOVL C02092 V=800.0 PL=0
MOVL C02093 V=800.0 PL=0
MOVL C02094 V=800.0 PL=0
MOVL C02095 V=800.0 PL=0
MOVL C02096 V=800.0 PL=0
MOVL C02097 V=800.0 PL=0
MOVL C02098 V=800.0 PL=0
MOVL C02099 V=800.0 PL=0
MOVL C02100 V=800.0 PL=0
MOVL C02101 V=800.0 PL=0
MOVL C02102 V=800.0 PL=0
MOVL C02103 V=800.0 PL=0
MOVL C02104 V=800.0 PL=0
MOVL C02105 V=800.0 PL=0
MOVL C02106 V=800.0 PL=0
MOVL C02107 V=800.0 PL=0
MOVL C02108 V=800.0 PL=0
MOVL C02109 V=800.0 PL=0
MOVL C02110 V=800.0 PL=0
MOVL C02111 V=800.0 PL=0
MOVL C02112 V=800.0 PL=0
MOVL C02113 V=800.0 PL=0
MOVL C02114 V=800.0 PL=0
MOVL C02115 V=800.0 PL=0
MOVL C02116 V=800.0 PL=0
MOVL C02117 V=800.0 PL=0
MOVL C02118 V=800.0 PL=0
MOVL C02119 V=800.0 PL=0
MOVL C02120 V=800.0 PL=0
MOVL C02121 V=800.0 PL=0
MOVL C02122 V=800.0 PL=0
MOVL C02123 V=800.0 PL=0
MOVL C02124 V=800.0 PL=0
MOVL C02125 V=800.0 PL=0
MOVL C02126 V=800.0 PL=0
MOVL C02127 V=800.0 PL=0
MOVL C02128 V=800.0 PL=0
MOVL C02129 V=800.0 PL=0
MOVL C02130 V=800.0 PL=0
MOVL C02131 V=800.0 PL=0
MOVL C02132 V=800.0 PL=0
MOVL C02133 V=800.0 PL=0
MOVL C02134 V=800.0 PL=0
MOVL C02135 V=800.0 PL=0
MOVL C02136 V=800.0 PL=0
MOVL C02137 V=800.0 PL=0
MOVL C02138 V=800.0 PL=0
MOVL C02139 V=800.0 PL=0
MOVL C02140 V=800.0 PL=0
MOVL C02141 V=800.0 PL=0
MOVL C02142 V=800.0 PL=0
MOVL C02143 V=800.0 PL=0
MOVL C02144 V=800.0 PL=0
MOVL C02145 V=800.0 PL=0
MOVL C02146 V=800.0 PL=0
MOVL C02147 V=800.0 PL=0
MOVL C02148 V=800.0 PL=0
MOVL C02149 V=800.0 PL=0
MOVL C02150 V=800.0 PL=0
